LIN {X 0,Y 523.912,Z 870.031,A -85,B 0,C 180,E1 -4697.971,E2 -4697.971} C_VEL
LIN {X 0,Y 523.923,Z 870.031,A -85,B 0,C 180,E1 -4700.412,E2 -4700.412} C_VEL
LIN {X 0,Y 523.884,Z 870.04,A -85,B 0,C 180,E1 -4702.895,E2 -4702.895} C_VEL
LIN {X 0,Y 523.871,Z 870.043,A -85,B 0,C 180,E1 -4705.423,E2 -4705.423} C_VEL
LIN {X 0,Y 523.896,Z 870.034,A -85,B 0,C 180,E1 -4708.003,E2 -4708.003} C_VEL
LIN {X 0,Y 523.895,Z 870.034,A -85,B 0,C 180,E1 -4710.845,E2 -4710.845} C_VEL
LIN {X 0,Y 523.911,Z 870.039,A -85,B 0,C 180,E1 -4713.726,E2 -4713.726} C_VEL
LIN {X 0,Y 523.854,Z 870.039,A -85,B 0,C 180,E1 -4716.393,E2 -4716.393} C_VEL
LIN {X 0,Y 523.886,Z 870.034,A -85,B 0,C 180,E1 -4719.088,E2 -4719.088} C_VEL
LIN {X 0,Y 523.885,Z 870.042,A -85,B 0,C 180,E1 -4722.125,E2 -4722.125} C_VEL
LIN {X 0,Y 523.93,Z 870.029,A -85,B 0,C 180,E1 -4725.311,E2 -4725.311} C_VEL
LIN {X 0,Y 523.875,Z 870.039,A -85,B 0,C 180,E1 -4728.7,E2 -4728.7} C_VEL
LIN {X 0,Y 523.872,Z 870.038,A -85,B 0,C 180,E1 -4731.894,E2 -4731.894} C_VEL
LIN {X 0,Y 523.912,Z 870.035,A -85,B 0,C 180,E1 -4734.913,E2 -4734.913} C_VEL
LIN {X 0,Y 523.899,Z 870.032,A -85,B 0,C 180,E1 -4737.686,E2 -4737.686} C_VEL
LIN {X 0,Y 523.864,Z 870.039,A -85,B 0,C 180,E1 -4740.239,E2 -4740.239} C_VEL
LIN {X 0,Y 523.889,Z 870.043,A -85,B 0,C 180,E1 -4742.863,E2 -4742.863} C_VEL
LIN {X 0,Y 523.909,Z 870.036,A -85,B 0,C 180,E1 -4745.809,E2 -4745.809} C_VEL
LIN {X 0,Y 523.951,Z 870.114,A -85,B 0,C 180,E1 -4746.821,E2 -4746.821} C_VEL
LIN {X 0,Y 525.037,Z 877.349,A -85,B 0,C 180,E1 -4748.194,E2 -4748.194} C_VEL
LIN {X 0,Y 524.713,Z 893.158,A -85,B 0,C 180,E1 -4751.046,E2 -4751.046} C_VEL
LIN {X 0,Y 524.282,Z 909.934,A -85,B 0,C 180,E1 -4754.05,E2 -4754.05} C_VEL
LIN {X 0,Y 523.984,Z 926.682,A -85,B 0,C 180,E1 -4757.017,E2 -4757.017} C_VEL
LIN {X 0,Y 523.894,Z 932.763,A -85,B 0,C 180,E1 -4758.086,E2 -4758.086} C_VEL
LIN {X 0,Y 524.95,Z 941.667,A -85,B 0,C 180,E1 -4758.233,E2 -4758.233} C_VEL
LIN {X 0,Y 524.777,Z 1009.129,A -85,B 0,C 180,E1 -4759.169,E2 -4759.169} C_VEL
LIN {X 0,Y 524.62,Z 1018.404,A -85,B 0,C 180,E1 -4759.385,E2 -4759.385} C_VEL
LIN {X 0,Y 524.516,Z 1026.88,A -85,B 0,C 180,E1 -4759.676,E2 -4759.676} C_VEL
LIN {X 0,Y 524.389,Z 1035.388,A -85,B 0,C 180,E1 -4760.063,E2 -4760.063} C_VEL
LIN {X 0,Y 524.242,Z 1043.722,A -85,B 0,C 180,E1 -4760.548,E2 -4760.548} C_VEL
LIN {X 0,Y 524.1,Z 1051.761,A -85,B 0,C 180,E1 -4761.129,E2 -4761.129} C_VEL
LIN {X 0,Y 523.896,Z 1060.43,A -85,B 0,C 180,E1 -4761.902,E2 -4761.902} C_VEL
LIN {X 0,Y 523.705,Z 1068.937,A -85,B 0,C 180,E1 -4762.869,E2 -4762.869} C_VEL
LIN {X 0,Y 523.627,Z 1075.609,A -85,B 0,C 180,E1 -4763.836,E2 -4763.836} C_VEL
LIN {X 0,Y 523.485,Z 1079.988,A -85,B 0,C 180,E1 -4764.607,E2 -4764.607} C_VEL
LIN {X 0,Y 523.469,Z 1085.148,A -85,B 0,C 180,E1 -4765.765,E2 -4765.765} C_VEL
LIN {X 0,Y 523.412,Z 1087.787,A -85,B 0,C 180,E1 -4766.536,E2 -4766.536} C_VEL
LIN {X 0,Y 523.336,Z 1090.682,A -85,B 0,C 180,E1 -4767.691,E2 -4767.691} C_VEL
LIN {X 0,Y 523.273,Z 1091.931,A -85,B 0,C 180,E1 -4768.461,E2 -4768.461} C_VEL
LIN {X 0,Y 523.246,Z 1092.708,A -85,B 0,C 180,E1 -4769.23,E2 -4769.23} C_VEL
LIN {X 0,Y 523.243,Z 1093,A -85,B 0,C 180,E1 -4770,E2 -4770} C_VEL
LIN {X 0,Y 523.246,Z 1092.707,A -85,B 0,C 180,E1 -4770.769,E2 -4770.769} C_VEL
LIN {X 0,Y 523.273,Z 1091.931,A -85,B 0,C 180,E1 -4771.539,E2 -4771.539} C_VEL
LIN {X 0,Y 523.335,Z 1090.681,A -85,B 0,C 180,E1 -4772.309,E2 -4772.309} C_VEL
LIN {X 0,Y 523.407,Z 1087.787,A -85,B 0,C 180,E1 -4773.464,E2 -4773.464} C_VEL
LIN {X 0,Y 523.472,Z 1085.149,A -85,B 0,C 180,E1 -4774.235,E2 -4774.235} C_VEL
LIN {X 0,Y 523.484,Z 1079.986,A -85,B 0,C 180,E1 -4775.392,E2 -4775.392} C_VEL
LIN {X 0,Y 523.667,Z 1073.736,A -85,B 0,C 180,E1 -4776.469,E2 -4776.469} C_VEL
LIN {X 0,Y 523.752,Z 1065.742,A -85,B 0,C 180,E1 -4777.517,E2 -4777.517} C_VEL
LIN {X 0,Y 523.93,Z 1058.402,A -85,B 0,C 180,E1 -4778.291,E2 -4778.291} C_VEL
LIN {X 0,Y 524.154,Z 1050.538,A -85,B 0,C 180,E1 -4778.967,E2 -4778.967} C_VEL
LIN {X 0,Y 524.246,Z 1042.226,A -85,B 0,C 180,E1 -4779.549,E2 -4779.549} C_VEL
LIN {X 0,Y 524.484,Z 1031.613,A -85,B 0,C 180,E1 -4780.129,E2 -4780.129} C_VEL
LIN {X 0,Y 524.584,Z 1020.08,A -85,B 0,C 180,E1 -4780.566,E2 -4780.566} C_VEL
LIN {X 0,Y 524.741,Z 1010.444,A -85,B 0,C 180,E1 -4780.807,E2 -4780.807} C_VEL
LIN {X 0,Y 524.94,Z 952.856,A -85,B 0,C 180,E1 -4781.614,E2 -4781.614} C_VEL
LIN {X 0,Y 524.776,Z 939.225,A -85,B 0,C 180,E1 -4781.804,E2 -4781.804} C_VEL
LIN {X 0,Y 523.913,Z 932.728,A -85,B 0,C 180,E1 -4781.92,E2 -4781.92} C_VEL
LIN {X 0,Y 524.196,Z 915.268,A -85,B 0,C 180,E1 -4785.001,E2 -4785.001} C_VEL
LIN {X 0,Y 524.626,Z 896.76,A -85,B 0,C 180,E1 -4788.309,E2 -4788.309} C_VEL
LIN {X 0,Y 524.982,Z 879.434,A -85,B 0,C 180,E1 -4791.395,E2 -4791.395} C_VEL
LIN {X 0,Y 524.731,Z 874.352,A -85,B 0,C 180,E1 -4792.321,E2 -4792.321} C_VEL
LIN {X 0,Y 523.943,Z 870.037,A -85,B 0,C 180,E1 -4793.153,E2 -4793.153} C_VEL
LIN {X 0,Y 523.876,Z 870.04,A -85,B 0,C 180,E1 -4796.277,E2 -4796.277} C_VEL
LIN {X 0,Y 523.869,Z 870.044,A -85,B 0,C 180,E1 -4798.879,E2 -4798.879} C_VEL
LIN {X 0,Y 523.902,Z 870.04,A -85,B 0,C 180,E1 -4801.545,E2 -4801.545} C_VEL
LIN {X 0,Y 523.908,Z 870.033,A -85,B 0,C 180,E1 -4804.292,E2 -4804.292} C_VEL
LIN {X 0,Y 523.845,Z 870.044,A -85,B 0,C 180,E1 -4807.137,E2 -4807.137} C_VEL
LIN {X 0,Y 523.88,Z 870.038,A -85,B 0,C 180,E1 -4810.122,E2 -4810.122} C_VEL
LIN {X 0,Y 523.869,Z 870.038,A -85,B 0,C 180,E1 -4813.172,E2 -4813.172} C_VEL
LIN {X 0,Y 523.912,Z 870.039,A -85,B 0,C 180,E1 -4815.769,E2 -4815.769} C_VEL
LIN {X 0,Y 523.851,Z 870.039,A -85,B 0,C 180,E1 -4818.899,E2 -4818.899} C_VEL
LIN {X 0,Y 523.871,Z 870.042,A -85,B 0,C 180,E1 -4821.895,E2 -4821.895} C_VEL
LIN {X 0,Y 523.911,Z 870.034,A -85,B 0,C 180,E1 -4824.913,E2 -4824.913} C_VEL
LIN {X 0,Y 523.898,Z 870.034,A -85,B 0,C 180,E1 -4827.686,E2 -4827.686} C_VEL
LIN {X 0,Y 523.863,Z 870.042,A -85,B 0,C 180,E1 -4830.239,E2 -4830.239} C_VEL
LIN {X 0,Y 523.888,Z 870.043,A -85,B 0,C 180,E1 -4832.864,E2 -4832.864} C_VEL
LIN {X 0,Y 523.899,Z 870.036,A -85,B 0,C 180,E1 -4835.812,E2 -4835.812} C_VEL
LIN {X 0,Y 523.914,Z 870.041,A -85,B 0,C 180,E1 -4838.766,E2 -4838.766} C_VEL
LIN {X 0,Y 523.915,Z 870.041,A -85,B 0,C 180,E1 -4841.22,E2 -4841.22} C_VEL
LIN {X 0,Y 523.957,Z 870.182,A -85,B 0,C 180,E1 -4842.311,E2 -4842.311} C_VEL
LIN {X 0,Y 523.897,Z 880.418,A -85,B 0,C 180,E1 -4844.783,E2 -4844.783} C_VEL
LIN {X 0,Y 523.686,Z 894.295,A -85,B 0,C 180,E1 -4848.063,E2 -4848.063} C_VEL
LIN {X 0,Y 523.712,Z 894.979,A -85,B 0,C 180,E1 -4848.158,E2 -4848.158} C_VEL
LIN {X 0,Y 524.962,Z 903.624,A -85,B 0,C 180,E1 -4848.305,E2 -4848.305} C_VEL
LIN {X 0,Y 524.729,Z 969.368,A -85,B 0,C 180,E1 -4849.217,E2 -4849.217} C_VEL
LIN {X 0,Y 524.665,Z 978.561,A -85,B 0,C 180,E1 -4849.436,E2 -4849.436} C_VEL
LIN {X 0,Y 524.486,Z 988.212,A -85,B 0,C 180,E1 -4849.773,E2 -4849.773} C_VEL
LIN {X 0,Y 524.359,Z 998.292,A -85,B 0,C 180,E1 -4850.258,E2 -4850.258} C_VEL
LIN {X 0,Y 524.191,Z 1008.741,A -85,B 0,C 180,E1 -4850.936,E2 -4850.936} C_VEL
LIN {X 0,Y 523.927,Z 1017.984,A -85,B 0,C 180,E1 -4851.709,E2 -4851.709} C_VEL
LIN {X 0,Y 523.774,Z 1025.419,A -85,B 0,C 180,E1 -4852.483,E2 -4852.483} C_VEL
LIN {X 0,Y 523.663,Z 1032.503,A -85,B 0,C 180,E1 -4853.4,E2 -4853.4} C_VEL
LIN {X 0,Y 523.545,Z 1038.794,A -85,B 0,C 180,E1 -4854.415,E2 -4854.415} C_VEL
LIN {X 0,Y 523.417,Z 1043.444,A -85,B 0,C 180,E1 -4855.379,E2 -4855.379} C_VEL
LIN {X 0,Y 523.408,Z 1047.699,A -85,B 0,C 180,E1 -4856.536,E2 -4856.536} C_VEL
LIN {X 0,Y 523.336,Z 1050.634,A -85,B 0,C 180,E1 -4857.691,E2 -4857.691} C_VEL
LIN {X 0,Y 523.273,Z 1051.934,A -85,B 0,C 180,E1 -4858.461,E2 -4858.461} C_VEL
LIN {X 0,Y 523.246,Z 1052.719,A -85,B 0,C 180,E1 -4859.231,E2 -4859.231} C_VEL
LIN {X 0,Y 523.244,Z 1052.997,A -85,B 0,C 180,E1 -4860,E2 -4860} C_VEL
LIN {X 0,Y 523.247,Z 1052.771,A -85,B 0,C 180,E1 -4860.77,E2 -4860.77} C_VEL
LIN {X 0,Y 523.274,Z 1052.046,A -85,B 0,C 180,E1 -4861.54,E2 -4861.54} C_VEL
LIN {X 0,Y 523.337,Z 1050.82,A -85,B 0,C 180,E1 -4862.309,E2 -4862.309} C_VEL
LIN {X 0,Y 523.406,Z 1047.96,A -85,B 0,C 180,E1 -4863.464,E2 -4863.464} C_VEL
LIN {X 0,Y 523.409,Z 1043.83,A -85,B 0,C 180,E1 -4864.621,E2 -4864.621} C_VEL
LIN {X 0,Y 523.606,Z 1038.224,A -85,B 0,C 180,E1 -4865.778,E2 -4865.778} C_VEL
LIN {X 0,Y 523.623,Z 1032.601,A -85,B 0,C 180,E1 -4866.676,E2 -4866.676} C_VEL
LIN {X 0,Y 523.789,Z 1024.48,A -85,B 0,C 180,E1 -4867.711,E2 -4867.711} C_VEL
LIN {X 0,Y 523.987,Z 1015.836,A -85,B 0,C 180,E1 -4868.582,E2 -4868.582} C_VEL
LIN {X 0,Y 524.228,Z 1005.965,A -85,B 0,C 180,E1 -4869.355,E2 -4869.355} C_VEL
LIN {X 0,Y 524.376,Z 996.263,A -85,B 0,C 180,E1 -4869.937,E2 -4869.937} C_VEL
LIN {X 0,Y 524.486,Z 988.005,A -85,B 0,C 180,E1 -4870.325,E2 -4870.325} C_VEL
LIN {X 0,Y 524.604,Z 979.109,A -85,B 0,C 180,E1 -4870.64,E2 -4870.64} C_VEL
LIN {X 0,Y 524.761,Z 970.227,A -85,B 0,C 180,E1 -4870.856,E2 -4870.856} C_VEL
LIN {X 0,Y 524.819,Z 902.474,A -85,B 0,C 180,E1 -4871.804,E2 -4871.804} C_VEL
LIN {X 0,Y 523.675,Z 894.664,A -85,B 0,C 180,E1 -4871.941,E2 -4871.941} C_VEL
LIN {X 0,Y 523.898,Z 880.793,A -85,B 0,C 180,E1 -4875.217,E2 -4875.217} C_VEL
LIN {X 0,Y 524.012,Z 870.024,A -85,B 0,C 180,E1 -4877.816,E2 -4877.816} C_VEL
LIN {X 0,Y 523.916,Z 870.038,A -85,B 0,C 180,E1 -4881.235,E2 -4881.235} C_VEL
LIN {X 0,Y 523.898,Z 870.034,A -85,B 0,C 180,E1 -4884.574,E2 -4884.574} C_VEL
LIN {X 0,Y 523.913,Z 870.036,A -85,B 0,C 180,E1 -4887.705,E2 -4887.705} C_VEL
LIN {X 0,Y 523.899,Z 870.034,A -85,B 0,C 180,E1 -4890.846,E2 -4890.846} C_VEL
LIN {X 0,Y 523.927,Z 870.037,A -85,B 0,C 180,E1 -4893.729,E2 -4893.729} C_VEL
LIN {X 0,Y 523.856,Z 870.04,A -85,B 0,C 180,E1 -4896.279,E2 -4896.279} C_VEL
LIN {X 0,Y 523.205,Z 870.12,A -85,B 0,C 180,E1 -4896.921,E2 -4896.921} C_VEL
LIN {X 0,Y 520.366,Z 870.48,A -85,B 0,C 180,E1 -4897.963,E2 -4897.963} C_VEL
LIN {X 0,Y 517.955,Z 870.776,A -85,B 0,C 180,E1 -4898.802,E2 -4898.802} C_VEL
LIN {X 0,Y 516.915,Z 870.906,A -85,B 0,C 180,E1 -4899.45,E2 -4899.45} C_VEL
LIN {X 0,Y 516.829,Z 870.919,A -85,B 0,C 180,E1 -4899.669,E2 -4899.669} C_VEL
LIN {X 0,Y 516.843,Z 870.912,A -85,B 0,C 180,E1 -4902.836,E2 -4902.836} C_VEL
LIN {X 0,Y 516.899,Z 870.905,A -85,B 0,C 180,E1 -4905.007,E2 -4905.007} C_VEL
LIN {X 0,Y 516.831,Z 870.921,A -85,B 0,C 180,E1 -4908.41,E2 -4908.41} C_VEL
LIN {X 0,Y 516.855,Z 870.91,A -85,B 0,C 180,E1 -4911.282,E2 -4911.282} C_VEL
LIN {X 0,Y 516.853,Z 870.918,A -85,B 0,C 180,E1 -4914.674,E2 -4914.674} C_VEL
LIN {X 0,Y 516.87,Z 870.909,A -85,B 0,C 180,E1 -4917.462,E2 -4917.462} C_VEL
LIN {X 0,Y 516.841,Z 870.916,A -85,B 0,C 180,E1 -4920.491,E2 -4920.491} C_VEL
LIN {X 0,Y 516.83,Z 870.917,A -85,B 0,C 180,E1 -4923.337,E2 -4923.337} C_VEL
LIN {X 0,Y 516.871,Z 870.908,A -85,B 0,C 180,E1 -4925.926,E2 -4925.926} C_VEL
LIN {X 0,Y 516.869,Z 870.909,A -85,B 0,C 180,E1 -4928.462,E2 -4928.462} C_VEL
LIN {X 0,Y 516.871,Z 870.912,A -85,B 0,C 180,E1 -4930.954,E2 -4930.954} C_VEL
LIN {X 0,Y 516.876,Z 870.917,A -85,B 0,C 180,E1 -4933.409,E2 -4933.409} C_VEL
LIN {X 0,Y 516.875,Z 870.912,A -85,B 0,C 180,E1 -4935.833,E2 -4935.833} C_VEL
LIN {X 0,Y 516.925,Z 870.903,A -85,B 0,C 180,E1 -4938.233,E2 -4938.233} C_VEL
LIN {X 0,Y 516.921,Z 870.906,A -85,B 0,C 180,E1 -4941.399,E2 -4941.399} C_VEL
LIN {X 0,Y 516.981,Z 870.896,A -85,B 0,C 180,E1 -4944.54,E2 -4944.54} C_VEL
LIN {X 0,Y 517.071,Z 870.887,A -85,B 0,C 180,E1 -4947.663,E2 -4947.663} C_VEL
LIN {X 0,Y 517.068,Z 870.891,A -85,B 0,C 180,E1 -4950,E2 -4950} C_VEL
LIN {X 0,Y 517.068,Z 870.891,A -85,B 0,C 180,E1 -4952.337,E2 -4952.337} C_VEL
LIN {X 0,Y 516.97,Z 870.903,A -85,B 0,C 180,E1 -4956.244,E2 -4956.244} C_VEL
LIN {X 0,Y 516.905,Z 870.904,A -85,B 0,C 180,E1 -4959.39,E2 -4959.39} C_VEL
LIN {X 0,Y 516.884,Z 870.914,A -85,B 0,C 180,E1 -4962.565,E2 -4962.565} C_VEL
LIN {X 0,Y 516.838,Z 870.912,A -85,B 0,C 180,E1 -4965.781,E2 -4965.781} C_VEL
LIN {X 0,Y 516.875,Z 870.908,A -85,B 0,C 180,E1 -4968.224,E2 -4968.224} C_VEL
LIN {X 0,Y 516.882,Z 870.911,A -85,B 0,C 180,E1 -4970.703,E2 -4970.703} C_VEL
LIN {X 0,Y 516.841,Z 870.92,A -85,B 0,C 180,E1 -4973.225,E2 -4973.225} C_VEL
LIN {X 0,Y 516.861,Z 870.909,A -85,B 0,C 180,E1 -4976.176,E2 -4976.176} C_VEL
LIN {X 0,Y 516.833,Z 870.913,A -85,B 0,C 180,E1 -4978.421,E2 -4978.421} C_VEL
LIN {X 0,Y 516.849,Z 870.914,A -85,B 0,C 180,E1 -4981.112,E2 -4981.112} C_VEL
LIN {X 0,Y 516.873,Z 870.913,A -85,B 0,C 180,E1 -4983.959,E2 -4983.959} C_VEL
LIN {X 0,Y 516.799,Z 870.917,A -85,B 0,C 180,E1 -4986.753,E2 -4986.753} C_VEL
LIN {X 0,Y 516.827,Z 870.921,A -85,B 0,C 180,E1 -4989.727,E2 -4989.727} C_VEL
LIN {X 0,Y 516.841,Z 870.912,A -85,B 0,C 180,E1 -4992.836,E2 -4992.836} C_VEL
LIN {X 0,Y 516.901,Z 870.904,A -85,B 0,C 180,E1 -4995.007,E2 -4995.007} C_VEL
LIN {X 0,Y 516.832,Z 870.92,A -85,B 0,C 180,E1 -4998.409,E2 -4998.409} C_VEL
LIN {X 0,Y 516.854,Z 870.91,A -85,B 0,C 180,E1 -5001.281,E2 -5001.281} C_VEL
LIN {X 0,Y 516.852,Z 870.918,A -85,B 0,C 180,E1 -5004.673,E2 -5004.673} C_VEL
LIN {X 0,Y 516.871,Z 870.909,A -85,B 0,C 180,E1 -5007.462,E2 -5007.462} C_VEL
LIN {X 0,Y 516.841,Z 870.916,A -85,B 0,C 180,E1 -5010.491,E2 -5010.491} C_VEL
LIN {X 0,Y 516.83,Z 870.917,A -85,B 0,C 180,E1 -5013.336,E2 -5013.336} C_VEL
LIN {X 0,Y 516.871,Z 870.908,A -85,B 0,C 180,E1 -5015.926,E2 -5015.926} C_VEL
LIN {X 0,Y 516.869,Z 870.909,A -85,B 0,C 180,E1 -5018.461,E2 -5018.461} C_VEL
LIN {X 0,Y 516.87,Z 870.913,A -85,B 0,C 180,E1 -5020.953,E2 -5020.953} C_VEL
LIN {X 0,Y 516.874,Z 870.917,A -85,B 0,C 180,E1 -5023.408,E2 -5023.408} C_VEL
LIN {X 0,Y 516.867,Z 870.913,A -85,B 0,C 180,E1 -5025.832,E2 -5025.832} C_VEL
LIN {X 0,Y 516.923,Z 870.903,A -85,B 0,C 180,E1 -5028.232,E2 -5028.232} C_VEL
LIN {X 0,Y 516.919,Z 870.906,A -85,B 0,C 180,E1 -5031.398,E2 -5031.398} C_VEL
LIN {X 0,Y 516.979,Z 870.896,A -85,B 0,C 180,E1 -5034.539,E2 -5034.539} C_VEL
LIN {X 0,Y 517.069,Z 870.888,A -85,B 0,C 180,E1 -5037.663,E2 -5037.663} C_VEL
LIN {X 0,Y 517.066,Z 870.892,A -85,B 0,C 180,E1 -5040,E2 -5040} C_VEL
LIN {X 0,Y 517.066,Z 870.891,A -85,B 0,C 180,E1 -5042.337,E2 -5042.337} C_VEL
LIN {X 0,Y 516.968,Z 870.903,A -85,B 0,C 180,E1 -5046.243,E2 -5046.243} C_VEL
LIN {X 0,Y 516.902,Z 870.904,A -85,B 0,C 180,E1 -5049.39,E2 -5049.39} C_VEL
LIN {X 0,Y 516.882,Z 870.915,A -85,B 0,C 180,E1 -5052.565,E2 -5052.565} C_VEL
LIN {X 0,Y 516.904,Z 870.908,A -85,B 0,C 180,E1 -5055.128,E2 -5055.128} C_VEL
LIN {X 0,Y 516.871,Z 870.909,A -85,B 0,C 180,E1 -5058.224,E2 -5058.224} C_VEL
LIN {X 0,Y 516.879,Z 870.912,A -85,B 0,C 180,E1 -5060.703,E2 -5060.703} C_VEL
LIN {X 0,Y 516.837,Z 870.921,A -85,B 0,C 180,E1 -5063.225,E2 -5063.225} C_VEL
LIN {X 0,Y 516.857,Z 870.91,A -85,B 0,C 180,E1 -5066.176,E2 -5066.176} C_VEL
LIN {X 0,Y 516.829,Z 870.913,A -85,B 0,C 180,E1 -5068.42,E2 -5068.42} C_VEL
LIN {X 0,Y 516.845,Z 870.915,A -85,B 0,C 180,E1 -5071.112,E2 -5071.112} C_VEL
LIN {X 0,Y 516.869,Z 870.913,A -85,B 0,C 180,E1 -5073.959,E2 -5073.959} C_VEL
LIN {X 0,Y 516.795,Z 870.917,A -85,B 0,C 180,E1 -5076.753,E2 -5076.753} C_VEL
LIN {X 0,Y 516.823,Z 870.922,A -85,B 0,C 180,E1 -5079.727,E2 -5079.727} C_VEL
LIN {X 0,Y 516.836,Z 870.913,A -85,B 0,C 180,E1 -5082.836,E2 -5082.836} C_VEL
LIN {X 0,Y 516.896,Z 870.905,A -85,B 0,C 180,E1 -5085.007,E2 -5085.007} C_VEL
LIN {X 0,Y 516.828,Z 870.92,A -85,B 0,C 180,E1 -5088.409,E2 -5088.409} C_VEL
LIN {X 0,Y 516.85,Z 870.911,A -85,B 0,C 180,E1 -5091.281,E2 -5091.281} C_VEL
LIN {X 0,Y 516.848,Z 870.918,A -85,B 0,C 180,E1 -5094.673,E2 -5094.673} C_VEL
LIN {X 0,Y 516.866,Z 870.909,A -85,B 0,C 180,E1 -5097.462,E2 -5097.462} C_VEL
LIN {X 0,Y 516.837,Z 870.917,A -85,B 0,C 180,E1 -5100.491,E2 -5100.491} C_VEL
LIN {X 0,Y 516.825,Z 870.921,A -85,B 0,C 180,E1 -5103.336,E2 -5103.336} C_VEL
LIN {X 0,Y 516.904,Z 870.951,A -85,B 0,C 180,E1 -5106.672,E2 -5106.672} C_VEL
LIN {X 0,Y 518.076,Z 878.33,A -85,B 0,C 180,E1 -5108.096,E2 -5108.096} C_VEL
LIN {X 0,Y 517.716,Z 894.138,A -85,B 0,C 180,E1 -5110.986,E2 -5110.986} C_VEL
LIN {X 0,Y 517.268,Z 912.167,A -85,B 0,C 180,E1 -5114.232,E2 -5114.232} C_VEL
LIN {X 0,Y 516.888,Z 930.032,A -85,B 0,C 180,E1 -5117.435,E2 -5117.435} C_VEL
LIN {X 0,Y 516.861,Z 932.914,A -85,B 0,C 180,E1 -5117.924,E2 -5117.924} C_VEL
LIN {X 0,Y 517.983,Z 941.173,A -85,B 0,C 180,E1 -5118.066,E2 -5118.066} C_VEL
LIN {X 0,Y 517.827,Z 1009.137,A -85,B 0,C 180,E1 -5119.022,E2 -5119.022} C_VEL
LIN {X 0,Y 517.654,Z 1018.404,A -85,B 0,C 180,E1 -5119.241,E2 -5119.241} C_VEL
LIN {X 0,Y 517.534,Z 1026.879,A -85,B 0,C 180,E1 -5119.535,E2 -5119.535} C_VEL
LIN {X 0,Y 517.4,Z 1035.386,A -85,B 0,C 180,E1 -5119.928,E2 -5119.928} C_VEL
LIN {X 0,Y 517.25,Z 1043.72,A -85,B 0,C 180,E1 -5120.419,E2 -5120.419} C_VEL
LIN {X 0,Y 517.098,Z 1051.759,A -85,B 0,C 180,E1 -5121.008,E2 -5121.008} C_VEL
LIN {X 0,Y 516.843,Z 1060.431,A -85,B 0,C 180,E1 -5121.791,E2 -5121.791} C_VEL
LIN {X 0,Y 516.655,Z 1068.937,A -85,B 0,C 180,E1 -5122.771,E2 -5122.771} C_VEL
LIN {X 0,Y 516.561,Z 1075.609,A -85,B 0,C 180,E1 -5123.751,E2 -5123.751} C_VEL
LIN {X 0,Y 516.431,Z 1079.988,A -85,B 0,C 180,E1 -5124.533,E2 -5124.533} C_VEL
LIN {X 0,Y 516.392,Z 1085.148,A -85,B 0,C 180,E1 -5125.707,E2 -5125.707} C_VEL
LIN {X 0,Y 516.329,Z 1087.787,A -85,B 0,C 180,E1 -5126.488,E2 -5126.488} C_VEL
LIN {X 0,Y 516.262,Z 1090.681,A -85,B 0,C 180,E1 -5127.659,E2 -5127.659} C_VEL
LIN {X 0,Y 516.19,Z 1091.93,A -85,B 0,C 180,E1 -5128.439,E2 -5128.439} C_VEL
LIN {X 0,Y 516.156,Z 1092.707,A -85,B 0,C 180,E1 -5129.22,E2 -5129.22} C_VEL
LIN {X 0,Y 516.151,Z 1093,A -85,B 0,C 180,E1 -5130,E2 -5130} C_VEL
LIN {X 0,Y 516.156,Z 1092.707,A -85,B 0,C 180,E1 -5130.78,E2 -5130.78} C_VEL
LIN {X 0,Y 516.19,Z 1091.93,A -85,B 0,C 180,E1 -5131.56,E2 -5131.56} C_VEL
LIN {X 0,Y 516.262,Z 1090.681,A -85,B 0,C 180,E1 -5132.34,E2 -5132.34} C_VEL
LIN {X 0,Y 516.325,Z 1087.787,A -85,B 0,C 180,E1 -5133.512,E2 -5133.512} C_VEL
LIN {X 0,Y 516.394,Z 1085.149,A -85,B 0,C 180,E1 -5134.293,E2 -5134.293} C_VEL
LIN {X 0,Y 516.431,Z 1079.986,A -85,B 0,C 180,E1 -5135.466,E2 -5135.466} C_VEL
LIN {X 0,Y 516.58,Z 1074.231,A -85,B 0,C 180,E1 -5136.478,E2 -5136.478} C_VEL
LIN {X 0,Y 516.683,Z 1067.436,A -85,B 0,C 180,E1 -5137.424,E2 -5137.424} C_VEL
LIN {X 0,Y 516.862,Z 1059.421,A -85,B 0,C 180,E1 -5138.307,E2 -5138.307} C_VEL
LIN {X 0,Y 517.07,Z 1051.767,A -85,B 0,C 180,E1 -5138.993,E2 -5138.993} C_VEL
LIN {X 0,Y 517.226,Z 1043.725,A -85,B 0,C 180,E1 -5139.581,E2 -5139.581} C_VEL
LIN {X 0,Y 517.399,Z 1035.393,A -85,B 0,C 180,E1 -5140.072,E2 -5140.072} C_VEL
LIN {X 0,Y 517.533,Z 1026.89,A -85,B 0,C 180,E1 -5140.465,E2 -5140.465} C_VEL
LIN {X 0,Y 517.689,Z 1016.753,A -85,B 0,C 180,E1 -5140.808,E2 -5140.808} C_VEL
LIN {X 0,Y 517.871,Z 1005.092,A -85,B 0,C 180,E1 -5141.051,E2 -5141.051} C_VEL
LIN {X 0,Y 517.887,Z 940.331,A -85,B 0,C 180,E1 -5141.948,E2 -5141.948} C_VEL
LIN {X 0,Y 516.853,Z 932.68,A -85,B 0,C 180,E1 -5142.093,E2 -5142.093} C_VEL
LIN {X 0,Y 517.199,Z 915.041,A -85,B 0,C 180,E1 -5145.25,E2 -5145.25} C_VEL
LIN {X 0,Y 517.609,Z 897.395,A -85,B 0,C 180,E1 -5148.402,E2 -5148.402} C_VEL
LIN {X 0,Y 517.903,Z 882.556,A -85,B 0,C 180,E1 -5151.076,E2 -5151.076} C_VEL
LIN {X 0,Y 517.904,Z 876.83,A -85,B 0,C 180,E1 -5152.121,E2 -5152.121} C_VEL
LIN {X 0,Y 516.884,Z 870.915,A -85,B 0,C 180,E1 -5153.276,E2 -5153.276} C_VEL
LIN {X 0,Y 516.824,Z 870.921,A -85,B 0,C 180,E1 -5156.663,E2 -5156.663} C_VEL
LIN {X 0,Y 516.835,Z 870.919,A -85,B 0,C 180,E1 -5159.509,E2 -5159.509} C_VEL
LIN {X 0,Y 516.864,Z 870.911,A -85,B 0,C 180,E1 -5162.538,E2 -5162.538} C_VEL
LIN {X 0,Y 516.846,Z 870.92,A -85,B 0,C 180,E1 -5165.327,E2 -5165.327} C_VEL
LIN {X 0,Y 516.848,Z 870.912,A -85,B 0,C 180,E1 -5168.719,E2 -5168.719} C_VEL
LIN {X 0,Y 516.828,Z 870.922,A -85,B 0,C 180,E1 -5171.784,E2 -5171.784} C_VEL
LIN {X 0,Y 516.894,Z 870.906,A -85,B 0,C 180,E1 -5175.007,E2 -5175.007} C_VEL
LIN {X 0,Y 516.827,Z 870.919,A -85,B 0,C 180,E1 -5178.41,E2 -5178.41} C_VEL
LIN {X 0,Y 516.849,Z 870.912,A -85,B 0,C 180,E1 -5181.282,E2 -5181.282} C_VEL
LIN {X 0,Y 516.847,Z 870.917,A -85,B 0,C 180,E1 -5184.674,E2 -5184.674} C_VEL
LIN {X 0,Y 516.865,Z 870.91,A -85,B 0,C 180,E1 -5187.462,E2 -5187.462} C_VEL
LIN {X 0,Y 516.836,Z 870.922,A -85,B 0,C 180,E1 -5190.491,E2 -5190.491} C_VEL
LIN {X 0,Y 516.824,Z 870.917,A -85,B 0,C 180,E1 -5193.337,E2 -5193.337} C_VEL
LIN {X 0,Y 516.856,Z 870.914,A -85,B 0,C 180,E1 -5195.926,E2 -5195.926} C_VEL
LIN {X 0,Y 516.858,Z 870.916,A -85,B 0,C 180,E1 -5198.461,E2 -5198.461} C_VEL
LIN {X 0,Y 516.865,Z 870.919,A -85,B 0,C 180,E1 -5200.954,E2 -5200.954} C_VEL
LIN {X 0,Y 516.889,Z 870.978,A -85,B 0,C 180,E1 -5202.186,E2 -5202.186} C_VEL
LIN {X 0,Y 516.911,Z 877.482,A -85,B 0,C 180,E1 -5203.816,E2 -5203.816} C_VEL
LIN {X 0,Y 516.712,Z 888.994,A -85,B 0,C 180,E1 -5206.631,E2 -5206.631} C_VEL
LIN {X 0,Y 516.642,Z 894.642,A -85,B 0,C 180,E1 -5207.98,E2 -5207.98} C_VEL
LIN {X 0,Y 518.042,Z 905.254,A -85,B 0,C 180,E1 -5208.169,E2 -5208.169} C_VEL
LIN {X 0,Y 517.755,Z 969.401,A -85,B 0,C 180,E1 -5209.07,E2 -5209.07} C_VEL
LIN {X 0,Y 517.697,Z 978.581,A -85,B 0,C 180,E1 -5209.292,E2 -5209.292} C_VEL
LIN {X 0,Y 517.512,Z 988.225,A -85,B 0,C 180,E1 -5209.634,E2 -5209.634} C_VEL
LIN {X 0,Y 517.371,Z 998.307,A -85,B 0,C 180,E1 -5210.125,E2 -5210.125} C_VEL
LIN {X 0,Y 517.169,Z 1008.744,A -85,B 0,C 180,E1 -5210.812,E2 -5210.812} C_VEL
LIN {X 0,Y 516.894,Z 1017.992,A -85,B 0,C 180,E1 -5211.596,E2 -5211.596} C_VEL
LIN {X 0,Y 516.712,Z 1025.429,A -85,B 0,C 180,E1 -5212.38,E2 -5212.38} C_VEL
LIN {X 0,Y 516.621,Z 1032.128,A -85,B 0,C 180,E1 -5213.255,E2 -5213.255} C_VEL
LIN {X 0,Y 516.496,Z 1038.797,A -85,B 0,C 180,E1 -5214.339,E2 -5214.339} C_VEL
LIN {X 0,Y 516.322,Z 1043.444,A -85,B 0,C 180,E1 -5215.316,E2 -5215.316} C_VEL
LIN {X 0,Y 516.326,Z 1047.704,A -85,B 0,C 180,E1 -5216.489,E2 -5216.489} C_VEL
LIN {X 0,Y 516.263,Z 1050.639,A -85,B 0,C 180,E1 -5217.66,E2 -5217.66} C_VEL
LIN {X 0,Y 516.19,Z 1051.937,A -85,B 0,C 180,E1 -5218.44,E2 -5218.44} C_VEL
LIN {X 0,Y 516.157,Z 1052.719,A -85,B 0,C 180,E1 -5219.22,E2 -5219.22} C_VEL
LIN {X 0,Y 516.152,Z 1052.997,A -85,B 0,C 180,E1 -5220,E2 -5220} C_VEL
LIN {X 0,Y 516.157,Z 1052.774,A -85,B 0,C 180,E1 -5220.781,E2 -5220.781} C_VEL
LIN {X 0,Y 516.191,Z 1052.05,A -85,B 0,C 180,E1 -5221.561,E2 -5221.561} C_VEL
LIN {X 0,Y 516.263,Z 1050.823,A -85,B 0,C 180,E1 -5222.341,E2 -5222.341} C_VEL
LIN {X 0,Y 516.324,Z 1047.959,A -85,B 0,C 180,E1 -5223.512,E2 -5223.512} C_VEL
LIN {X 0,Y 516.315,Z 1043.825,A -85,B 0,C 180,E1 -5224.685,E2 -5224.685} C_VEL
LIN {X 0,Y 516.553,Z 1038.221,A -85,B 0,C 180,E1 -5225.857,E2 -5225.857} C_VEL
LIN {X 0,Y 516.585,Z 1031.97,A -85,B 0,C 180,E1 -5226.86,E2 -5226.86} C_VEL
LIN {X 0,Y 516.735,Z 1024.473,A -85,B 0,C 180,E1 -5227.817,E2 -5227.817} C_VEL
LIN {X 0,Y 516.972,Z 1015.828,A -85,B 0,C 180,E1 -5228.699,E2 -5228.699} C_VEL
LIN {X 0,Y 517.203,Z 1005.953,A -85,B 0,C 180,E1 -5229.484,E2 -5229.484} C_VEL
LIN {X 0,Y 517.382,Z 996.248,A -85,B 0,C 180,E1 -5230.073,E2 -5230.073} C_VEL
LIN {X 0,Y 517.514,Z 987.987,A -85,B 0,C 180,E1 -5230.466,E2 -5230.466} C_VEL
LIN {X 0,Y 517.649,Z 979.087,A -85,B 0,C 180,E1 -5230.784,E2 -5230.784} C_VEL
LIN {X 0,Y 517.809,Z 970.348,A -85,B 0,C 180,E1 -5231.001,E2 -5231.001} C_VEL
LIN {X 0,Y 517.901,Z 903.29,A -85,B 0,C 180,E1 -5231.952,E2 -5231.952} C_VEL
LIN {X 0,Y 516.624,Z 894.661,A -85,B 0,C 180,E1 -5232.106,E2 -5232.106} C_VEL
LIN {X 0,Y 516.875,Z 881.245,A -85,B 0,C 180,E1 -5235.336,E2 -5235.336} C_VEL
LIN {X 0,Y 516.954,Z 870.904,A -85,B 0,C 180,E1 -5237.889,E2 -5237.889} C_VEL
LIN {X 0,Y 516.879,Z 870.911,A -85,B 0,C 180,E1 -5240.703,E2 -5240.703} C_VEL
LIN {X 0,Y 516.84,Z 870.921,A -85,B 0,C 180,E1 -5243.225,E2 -5243.225} C_VEL
LIN {X 0,Y 516.861,Z 870.909,A -85,B 0,C 180,E1 -5246.177,E2 -5246.177} C_VEL
LIN {X 0,Y 516.83,Z 870.913,A -85,B 0,C 180,E1 -5248.421,E2 -5248.421} C_VEL
LIN {X 0,Y 516.849,Z 870.914,A -85,B 0,C 180,E1 -5251.113,E2 -5251.113} C_VEL
LIN {X 0,Y 516.882,Z 870.912,A -85,B 0,C 180,E1 -5253.962,E2 -5253.962} C_VEL
LIN {X 0,Y 516.807,Z 870.916,A -85,B 0,C 180,E1 -5256.752,E2 -5256.752} C_VEL
LIN {X 0,Y 516.829,Z 870.919,A -85,B 0,C 180,E1 -5259.669,E2 -5259.669} C_VEL
LIN {X 0,Y 516.16,Z 871.009,A -85,B 0,C 180,E1 -5260.32,E2 -5260.32} C_VEL
LIN {X 0,Y 513.312,Z 871.362,A -85,B 0,C 180,E1 -5261.377,E2 -5261.377} C_VEL
LIN {X 0,Y 510.907,Z 871.657,A -85,B 0,C 180,E1 -5262.228,E2 -5262.228} C_VEL
LIN {X 0,Y 509.873,Z 871.78,A -85,B 0,C 180,E1 -5262.885,E2 -5262.885} C_VEL
LIN {X 0,Y 509.787,Z 871.791,A -85,B 0,C 180,E1 -5263.108,E2 -5263.108} C_VEL
LIN {X 0,Y 509.809,Z 871.792,A -85,B 0,C 180,E1 -5265.796,E2 -5265.796} C_VEL
LIN {X 0,Y 509.785,Z 871.796,A -85,B 0,C 180,E1 -5268.567,E2 -5268.567} C_VEL
LIN {X 0,Y 509.806,Z 871.789,A -85,B 0,C 180,E1 -5271.794,E2 -5271.794} C_VEL
LIN {X 0,Y 509.81,Z 871.796,A -85,B 0,C 180,E1 -5274.62,E2 -5274.62} C_VEL
LIN {X 0,Y 509.838,Z 871.785,A -85,B 0,C 180,E1 -5277.479,E2 -5277.479} C_VEL
LIN {X 0,Y 509.788,Z 871.793,A -85,B 0,C 180,E1 -5280.289,E2 -5280.289} C_VEL
LIN {X 0,Y 509.816,Z 871.796,A -85,B 0,C 180,E1 -5282.94,E2 -5282.94} C_VEL
LIN {X 0,Y 509.822,Z 871.789,A -85,B 0,C 180,E1 -5285.572,E2 -5285.572} C_VEL
LIN {X 0,Y 509.813,Z 871.787,A -85,B 0,C 180,E1 -5288.148,E2 -5288.148} C_VEL
LIN {X 0,Y 509.832,Z 871.786,A -85,B 0,C 180,E1 -5290.68,E2 -5290.68} C_VEL
LIN {X 0,Y 509.849,Z 871.789,A -85,B 0,C 180,E1 -5293.174,E2 -5293.174} C_VEL
LIN {X 0,Y 509.849,Z 871.79,A -85,B 0,C 180,E1 -5295.634,E2 -5295.634} C_VEL
LIN {X 0,Y 509.859,Z 871.782,A -85,B 0,C 180,E1 -5298.873,E2 -5298.873} C_VEL
LIN {X 0,Y 509.878,Z 871.784,A -85,B 0,C 180,E1 -5302.077,E2 -5302.077} C_VEL
LIN {X 0,Y 509.937,Z 871.774,A -85,B 0,C 180,E1 -5304.464,E2 -5304.464} C_VEL
LIN {X 0,Y 510.038,Z 871.763,A -85,B 0,C 180,E1 -5307.631,E2 -5307.631} C_VEL
LIN {X 0,Y 510.037,Z 871.767,A -85,B 0,C 180,E1 -5310,E2 -5310} C_VEL
LIN {X 0,Y 510.036,Z 871.767,A -85,B 0,C 180,E1 -5312.369,E2 -5312.369} C_VEL
LIN {X 0,Y 509.936,Z 871.772,A -85,B 0,C 180,E1 -5315.536,E2 -5315.536} C_VEL
LIN {X 0,Y 509.879,Z 871.781,A -85,B 0,C 180,E1 -5317.923,E2 -5317.923} C_VEL
LIN {X 0,Y 509.86,Z 871.784,A -85,B 0,C 180,E1 -5321.127,E2 -5321.127} C_VEL
LIN {X 0,Y 509.819,Z 871.787,A -85,B 0,C 180,E1 -5323.553,E2 -5323.553} C_VEL
LIN {X 0,Y 509.806,Z 871.788,A -85,B 0,C 180,E1 -5326.005,E2 -5326.005} C_VEL
LIN {X 0,Y 509.831,Z 871.788,A -85,B 0,C 180,E1 -5328.485,E2 -5328.485} C_VEL
LIN {X 0,Y 509.828,Z 871.794,A -85,B 0,C 180,E1 -5331.003,E2 -5331.003} C_VEL
LIN {X 0,Y 509.801,Z 871.793,A -85,B 0,C 180,E1 -5333.565,E2 -5333.565} C_VEL
LIN {X 0,Y 509.801,Z 871.789,A -85,B 0,C 180,E1 -5336.352,E2 -5336.352} C_VEL
LIN {X 0,Y 509.797,Z 871.791,A -85,B 0,C 180,E1 -5338.849,E2 -5338.849} C_VEL
LIN {X 0,Y 509.785,Z 871.799,A -85,B 0,C 180,E1 -5341.593,E2 -5341.593} C_VEL
LIN {X 0,Y 509.826,Z 871.786,A -85,B 0,C 180,E1 -5344.416,E2 -5344.416} C_VEL
LIN {X 0,Y 509.762,Z 871.797,A -85,B 0,C 180,E1 -5347.346,E2 -5347.346} C_VEL
LIN {X 0,Y 509.79,Z 871.793,A -85,B 0,C 180,E1 -5350.387,E2 -5350.387} C_VEL
LIN {X 0,Y 509.795,Z 871.792,A -85,B 0,C 180,E1 -5353.575,E2 -5353.575} C_VEL
LIN {X 0,Y 509.795,Z 871.795,A -85,B 0,C 180,E1 -5356.425,E2 -5356.425} C_VEL
LIN {X 0,Y 509.789,Z 871.791,A -85,B 0,C 180,E1 -5359.612,E2 -5359.612} C_VEL
LIN {X 0,Y 509.762,Z 871.8,A -85,B 0,C 180,E1 -5362.654,E2 -5362.654} C_VEL
LIN {X 0,Y 509.842,Z 871.784,A -85,B 0,C 180,E1 -5365.8,E2 -5365.8} C_VEL
LIN {X 0,Y 509.818,Z 871.796,A -85,B 0,C 180,E1 -5368.726,E2 -5368.726} C_VEL
LIN {X 0,Y 509.826,Z 871.786,A -85,B 0,C 180,E1 -5372.05,E2 -5372.05} C_VEL
LIN {X 0,Y 509.785,Z 871.796,A -85,B 0,C 180,E1 -5374.699,E2 -5374.699} C_VEL
LIN {X 0,Y 509.828,Z 871.79,A -85,B 0,C 180,E1 -5377.459,E2 -5377.459} C_VEL
LIN {X 0,Y 509.848,Z 871.784,A -85,B 0,C 180,E1 -5379.841,E2 -5379.841} C_VEL
LIN {X 0,Y 509.848,Z 871.789,A -85,B 0,C 180,E1 -5383.173,E2 -5383.173} C_VEL
LIN {X 0,Y 509.834,Z 871.792,A -85,B 0,C 180,E1 -5385.633,E2 -5385.633} C_VEL
LIN {X 0,Y 509.891,Z 871.78,A -85,B 0,C 180,E1 -5388.131,E2 -5388.131} C_VEL
LIN {X 0,Y 509.872,Z 871.783,A -85,B 0,C 180,E1 -5391.279,E2 -5391.279} C_VEL
LIN {X 0,Y 509.919,Z 871.781,A -85,B 0,C 180,E1 -5393.669,E2 -5393.669} C_VEL
LIN {X 0,Y 509.858,Z 871.782,A -85,B 0,C 180,E1 -5396.839,E2 -5396.839} C_VEL
LIN {X 0,Y 509.922,Z 871.778,A -85,B 0,C 180,E1 -5398.42,E2 -5398.42} C_VEL
LIN {X 0,Y 510.035,Z 871.768,A -85,B 0,C 180,E1 -5400,E2 -5400} C_VEL
LIN {X 0,Y 510.034,Z 871.767,A -85,B 0,C 180,E1 -5402.369,E2 -5402.369} C_VEL
LIN {X 0,Y 509.934,Z 871.772,A -85,B 0,C 180,E1 -5405.536,E2 -5405.536} C_VEL
LIN {X 0,Y 509.876,Z 871.781,A -85,B 0,C 180,E1 -5407.922,E2 -5407.922} C_VEL
LIN {X 0,Y 509.857,Z 871.784,A -85,B 0,C 180,E1 -5411.126,E2 -5411.126} C_VEL
LIN {X 0,Y 509.823,Z 871.786,A -85,B 0,C 180,E1 -5413.553,E2 -5413.553} C_VEL
LIN {X 0,Y 509.805,Z 871.788,A -85,B 0,C 180,E1 -5416.004,E2 -5416.004} C_VEL
LIN {X 0,Y 509.828,Z 871.788,A -85,B 0,C 180,E1 -5418.485,E2 -5418.485} C_VEL
LIN {X 0,Y 509.824,Z 871.795,A -85,B 0,C 180,E1 -5421.002,E2 -5421.002} C_VEL
LIN {X 0,Y 509.798,Z 871.793,A -85,B 0,C 180,E1 -5423.565,E2 -5423.565} C_VEL
LIN {X 0,Y 509.798,Z 871.789,A -85,B 0,C 180,E1 -5426.352,E2 -5426.352} C_VEL
LIN {X 0,Y 509.793,Z 871.792,A -85,B 0,C 180,E1 -5428.849,E2 -5428.849} C_VEL
LIN {X 0,Y 509.781,Z 871.799,A -85,B 0,C 180,E1 -5431.593,E2 -5431.593} C_VEL
LIN {X 0,Y 509.821,Z 871.787,A -85,B 0,C 180,E1 -5434.415,E2 -5434.415} C_VEL
LIN {X 0,Y 509.759,Z 871.797,A -85,B 0,C 180,E1 -5437.345,E2 -5437.345} C_VEL
LIN {X 0,Y 509.785,Z 871.794,A -85,B 0,C 180,E1 -5440.387,E2 -5440.387} C_VEL
LIN {X 0,Y 509.79,Z 871.793,A -85,B 0,C 180,E1 -5443.575,E2 -5443.575} C_VEL
LIN {X 0,Y 509.79,Z 871.796,A -85,B 0,C 180,E1 -5446.425,E2 -5446.425} C_VEL
LIN {X 0,Y 509.785,Z 871.792,A -85,B 0,C 180,E1 -5449.612,E2 -5449.612} C_VEL
LIN {X 0,Y 509.757,Z 871.8,A -85,B 0,C 180,E1 -5452.654,E2 -5452.654} C_VEL
LIN {X 0,Y 509.837,Z 871.785,A -85,B 0,C 180,E1 -5455.8,E2 -5455.8} C_VEL
LIN {X 0,Y 509.814,Z 871.797,A -85,B 0,C 180,E1 -5458.726,E2 -5458.726} C_VEL
LIN {X 0,Y 509.821,Z 871.786,A -85,B 0,C 180,E1 -5462.05,E2 -5462.05} C_VEL
LIN {X 0,Y 509.781,Z 871.801,A -85,B 0,C 180,E1 -5464.699,E2 -5464.699} C_VEL
LIN {X 0,Y 509.865,Z 871.93,A -85,B 0,C 180,E1 -5466.546,E2 -5466.546} C_VEL
LIN {X 0,Y 511.078,Z 879.309,A -85,B 0,C 180,E1 -5467.993,E2 -5467.993} C_VEL
LIN {X 0,Y 510.724,Z 895.118,A -85,B 0,C 180,E1 -5470.924,E2 -5470.924} C_VEL
LIN {X 0,Y 510.253,Z 913.083,A -85,B 0,C 180,E1 -5474.202,E2 -5474.202} C_VEL
LIN {X 0,Y 509.837,Z 931.036,A -85,B 0,C 180,E1 -5477.44,E2 -5477.44} C_VEL
LIN {X 0,Y 509.803,Z 932.766,A -85,B 0,C 180,E1 -5477.752,E2 -5477.752} C_VEL
LIN {X 0,Y 511.064,Z 943.143,A -85,B 0,C 180,E1 -5477.929,E2 -5477.929} C_VEL
LIN {X 0,Y 510.881,Z 1009.214,A -85,B 0,C 180,E1 -5478.872,E2 -5478.872} C_VEL
LIN {X 0,Y 510.696,Z 1018.403,A -85,B 0,C 180,E1 -5479.092,E2 -5479.092} C_VEL
LIN {X 0,Y 510.567,Z 1026.878,A -85,B 0,C 180,E1 -5479.391,E2 -5479.391} C_VEL
LIN {X 0,Y 510.414,Z 1035.384,A -85,B 0,C 180,E1 -5479.789,E2 -5479.789} C_VEL
LIN {X 0,Y 510.258,Z 1043.719,A -85,B 0,C 180,E1 -5480.286,E2 -5480.286} C_VEL
LIN {X 0,Y 510.087,Z 1051.757,A -85,B 0,C 180,E1 -5480.883,E2 -5480.883} C_VEL
LIN {X 0,Y 509.819,Z 1060.431,A -85,B 0,C 180,E1 -5481.677,E2 -5481.677} C_VEL
LIN {X 0,Y 509.606,Z 1068.937,A -85,B 0,C 180,E1 -5482.671,E2 -5482.671} C_VEL
LIN {X 0,Y 509.492,Z 1075.609,A -85,B 0,C 180,E1 -5483.664,E2 -5483.664} C_VEL
LIN {X 0,Y 509.382,Z 1079.988,A -85,B 0,C 180,E1 -5484.458,E2 -5484.458} C_VEL
LIN {X 0,Y 509.298,Z 1085.149,A -85,B 0,C 180,E1 -5485.647,E2 -5485.647} C_VEL
LIN {X 0,Y 509.251,Z 1087.786,A -85,B 0,C 180,E1 -5486.439,E2 -5486.439} C_VEL
LIN {X 0,Y 509.191,Z 1090.68,A -85,B 0,C 180,E1 -5487.627,E2 -5487.627} C_VEL
LIN {X 0,Y 509.111,Z 1091.929,A -85,B 0,C 180,E1 -5488.418,E2 -5488.418} C_VEL
LIN {X 0,Y 509.07,Z 1092.706,A -85,B 0,C 180,E1 -5489.209,E2 -5489.209} C_VEL
LIN {X 0,Y 509.062,Z 1093,A -85,B 0,C 180,E1 -5490,E2 -5490} C_VEL
LIN {X 0,Y 509.07,Z 1092.706,A -85,B 0,C 180,E1 -5490.791,E2 -5490.791} C_VEL
LIN {X 0,Y 509.111,Z 1091.929,A -85,B 0,C 180,E1 -5491.582,E2 -5491.582} C_VEL
LIN {X 0,Y 509.191,Z 1090.68,A -85,B 0,C 180,E1 -5492.373,E2 -5492.373} C_VEL
LIN {X 0,Y 509.247,Z 1087.787,A -85,B 0,C 180,E1 -5493.56,E2 -5493.56} C_VEL
LIN {X 0,Y 509.3,Z 1085.149,A -85,B 0,C 180,E1 -5494.353,E2 -5494.353} C_VEL
LIN {X 0,Y 509.382,Z 1079.986,A -85,B 0,C 180,E1 -5495.542,E2 -5495.542} C_VEL
LIN {X 0,Y 509.493,Z 1074.853,A -85,B 0,C 180,E1 -5496.463,E2 -5496.463} C_VEL
LIN {X 0,Y 509.619,Z 1067.436,A -85,B 0,C 180,E1 -5497.528,E2 -5497.528} C_VEL
LIN {X 0,Y 509.843,Z 1059.42,A -85,B 0,C 180,E1 -5498.422,E2 -5498.422} C_VEL
LIN {X 0,Y 510.053,Z 1051.765,A -85,B 0,C 180,E1 -5499.117,E2 -5499.117} C_VEL
LIN {X 0,Y 510.233,Z 1043.724,A -85,B 0,C 180,E1 -5499.714,E2 -5499.714} C_VEL
LIN {X 0,Y 510.414,Z 1035.392,A -85,B 0,C 180,E1 -5500.211,E2 -5500.211} C_VEL
LIN {X 0,Y 510.564,Z 1026.888,A -85,B 0,C 180,E1 -5500.609,E2 -5500.609} C_VEL
LIN {X 0,Y 510.738,Z 1016.753,A -85,B 0,C 180,E1 -5500.957,E2 -5500.957} C_VEL
LIN {X 0,Y 510.923,Z 1005.447,A -85,B 0,C 180,E1 -5501.198,E2 -5501.198} C_VEL
LIN {X 0,Y 511.01,Z 941.466,A -85,B 0,C 180,E1 -5502.096,E2 -5502.096} C_VEL
LIN {X 0,Y 509.835,Z 932.658,A -85,B 0,C 180,E1 -5502.266,E2 -5502.266} C_VEL
LIN {X 0,Y 510.154,Z 915.431,A -85,B 0,C 180,E1 -5505.349,E2 -5505.349} C_VEL
LIN {X 0,Y 510.59,Z 898.205,A -85,B 0,C 180,E1 -5508.456,E2 -5508.456} C_VEL
LIN {X 0,Y 510.999,Z 881.106,A -85,B 0,C 180,E1 -5511.586,E2 -5511.586} C_VEL
LIN {X 0,Y 510.729,Z 876.511,A -85,B 0,C 180,E1 -5512.449,E2 -5512.449} C_VEL
LIN {X 0,Y 509.847,Z 871.791,A -85,B 0,C 180,E1 -5513.401,E2 -5513.401} C_VEL
LIN {X 0,Y 509.795,Z 871.795,A -85,B 0,C 180,E1 -5516.352,E2 -5516.352} C_VEL
LIN {X 0,Y 509.79,Z 871.798,A -85,B 0,C 180,E1 -5518.85,E2 -5518.85} C_VEL
LIN {X 0,Y 509.786,Z 871.798,A -85,B 0,C 180,E1 -5521.592,E2 -5521.592} C_VEL
LIN {X 0,Y 509.83,Z 871.787,A -85,B 0,C 180,E1 -5524.415,E2 -5524.415} C_VEL
LIN {X 0,Y 509.756,Z 871.802,A -85,B 0,C 180,E1 -5527.346,E2 -5527.346} C_VEL
LIN {X 0,Y 509.783,Z 871.792,A -85,B 0,C 180,E1 -5530.388,E2 -5530.388} C_VEL
LIN {X 0,Y 509.788,Z 871.797,A -85,B 0,C 180,E1 -5533.575,E2 -5533.575} C_VEL
LIN {X 0,Y 509.788,Z 871.794,A -85,B 0,C 180,E1 -5536.425,E2 -5536.425} C_VEL
LIN {X 0,Y 509.783,Z 871.794,A -85,B 0,C 180,E1 -5539.613,E2 -5539.613} C_VEL
LIN {X 0,Y 509.757,Z 871.799,A -85,B 0,C 180,E1 -5542.654,E2 -5542.654} C_VEL
LIN {X 0,Y 509.836,Z 871.787,A -85,B 0,C 180,E1 -5545.801,E2 -5545.801} C_VEL
LIN {X 0,Y 509.813,Z 871.795,A -85,B 0,C 180,E1 -5548.726,E2 -5548.726} C_VEL
LIN {X 0,Y 509.82,Z 871.789,A -85,B 0,C 180,E1 -5552.05,E2 -5552.05} C_VEL
LIN {X 0,Y 509.779,Z 871.802,A -85,B 0,C 180,E1 -5554.699,E2 -5554.699} C_VEL
LIN {X 0,Y 509.822,Z 871.792,A -85,B 0,C 180,E1 -5557.459,E2 -5557.459} C_VEL
LIN {X 0,Y 509.826,Z 871.793,A -85,B 0,C 180,E1 -5560.68,E2 -5560.68} C_VEL
LIN {X 0,Y 509.867,Z 871.826,A -85,B 0,C 180,E1 -5562.071,E2 -5562.071} C_VEL
LIN {X 0,Y 509.938,Z 877.806,A -85,B 0,C 180,E1 -5563.589,E2 -5563.589} C_VEL
LIN {X 0,Y 509.69,Z 889.236,A -85,B 0,C 180,E1 -5566.444,E2 -5566.444} C_VEL
LIN {X 0,Y 509.615,Z 894.776,A -85,B 0,C 180,E1 -5567.812,E2 -5567.812} C_VEL
LIN {X 0,Y 511.101,Z 905.25,A -85,B 0,C 180,E1 -5568.006,E2 -5568.006} C_VEL
LIN {X 0,Y 510.806,Z 969.433,A -85,B 0,C 180,E1 -5568.92,E2 -5568.92} C_VEL
LIN {X 0,Y 510.709,Z 978.601,A -85,B 0,C 180,E1 -5569.143,E2 -5569.143} C_VEL
LIN {X 0,Y 510.537,Z 988.239,A -85,B 0,C 180,E1 -5569.491,E2 -5569.491} C_VEL
LIN {X 0,Y 510.379,Z 998.323,A -85,B 0,C 180,E1 -5569.989,E2 -5569.989} C_VEL
LIN {X 0,Y 510.193,Z 1007.417,A -85,B 0,C 180,E1 -5570.586,E2 -5570.586} C_VEL
LIN {X 0,Y 509.898,Z 1016.996,A -85,B 0,C 180,E1 -5571.38,E2 -5571.38} C_VEL
LIN {X 0,Y 509.668,Z 1025.435,A -85,B 0,C 180,E1 -5572.274,E2 -5572.274} C_VEL
LIN {X 0,Y 509.544,Z 1032.756,A -85,B 0,C 180,E1 -5573.255,E2 -5573.255} C_VEL
LIN {X 0,Y 509.429,Z 1038.8,A -85,B 0,C 180,E1 -5574.26,E2 -5574.26} C_VEL
LIN {X 0,Y 509.235,Z 1043.444,A -85,B 0,C 180,E1 -5575.25,E2 -5575.25} C_VEL
LIN {X 0,Y 509.248,Z 1047.707,A -85,B 0,C 180,E1 -5576.44,E2 -5576.44} C_VEL
LIN {X 0,Y 509.192,Z 1050.642,A -85,B 0,C 180,E1 -5577.627,E2 -5577.627} C_VEL
LIN {X 0,Y 509.111,Z 1051.937,A -85,B 0,C 180,E1 -5578.418,E2 -5578.418} C_VEL
LIN {X 0,Y 509.07,Z 1052.718,A -85,B 0,C 180,E1 -5579.209,E2 -5579.209} C_VEL
LIN {X 0,Y 509.063,Z 1052.997,A -85,B 0,C 180,E1 -5580,E2 -5580} C_VEL
LIN {X 0,Y 509.071,Z 1052.776,A -85,B 0,C 180,E1 -5580.791,E2 -5580.791} C_VEL
LIN {X 0,Y 509.112,Z 1052.054,A -85,B 0,C 180,E1 -5581.582,E2 -5581.582} C_VEL
LIN {X 0,Y 509.192,Z 1050.826,A -85,B 0,C 180,E1 -5582.373,E2 -5582.373} C_VEL
LIN {X 0,Y 509.246,Z 1047.958,A -85,B 0,C 180,E1 -5583.561,E2 -5583.561} C_VEL
LIN {X 0,Y 509.228,Z 1043.819,A -85,B 0,C 180,E1 -5584.75,E2 -5584.75} C_VEL
LIN {X 0,Y 509.491,Z 1038.217,A -85,B 0,C 180,E1 -5585.939,E2 -5585.939} C_VEL
LIN {X 0,Y 509.523,Z 1031.888,A -85,B 0,C 180,E1 -5586.966,E2 -5586.966} C_VEL
LIN {X 0,Y 509.698,Z 1024.466,A -85,B 0,C 180,E1 -5587.926,E2 -5587.926} C_VEL
LIN {X 0,Y 509.944,Z 1015.819,A -85,B 0,C 180,E1 -5588.82,E2 -5588.82} C_VEL
LIN {X 0,Y 510.21,Z 1005.94,A -85,B 0,C 180,E1 -5589.615,E2 -5589.615} C_VEL
LIN {X 0,Y 510.397,Z 996.233,A -85,B 0,C 180,E1 -5590.212,E2 -5590.212} C_VEL
LIN {X 0,Y 510.547,Z 987.969,A -85,B 0,C 180,E1 -5590.61,E2 -5590.61} C_VEL
LIN {X 0,Y 510.702,Z 979.064,A -85,B 0,C 180,E1 -5590.933,E2 -5590.933} C_VEL
LIN {X 0,Y 510.857,Z 970.439,A -85,B 0,C 180,E1 -5591.15,E2 -5591.15} C_VEL
LIN {X 0,Y 510.932,Z 903.651,A -85,B 0,C 180,E1 -5592.111,E2 -5592.111} C_VEL
LIN {X 0,Y 509.593,Z 894.741,A -85,B 0,C 180,E1 -5592.276,E2 -5592.276} C_VEL
LIN {X 0,Y 509.848,Z 881.444,A -85,B 0,C 180,E1 -5595.552,E2 -5595.552} C_VEL
LIN {X 0,Y 509.919,Z 871.842,A -85,B 0,C 180,E1 -5597.931,E2 -5597.931} C_VEL
LIN {X 0,Y 509.824,Z 871.795,A -85,B 0,C 180,E1 -5601.003,E2 -5601.003} C_VEL
LIN {X 0,Y 509.803,Z 871.793,A -85,B 0,C 180,E1 -5603.565,E2 -5603.565} C_VEL
LIN {X 0,Y 509.802,Z 871.789,A -85,B 0,C 180,E1 -5606.353,E2 -5606.353} C_VEL
LIN {X 0,Y 509.794,Z 871.791,A -85,B 0,C 180,E1 -5608.85,E2 -5608.85} C_VEL
LIN {X 0,Y 509.79,Z 871.799,A -85,B 0,C 180,E1 -5611.593,E2 -5611.593} C_VEL
LIN {X 0,Y 509.834,Z 871.785,A -85,B 0,C 180,E1 -5614.415,E2 -5614.415} C_VEL
LIN {X 0,Y 509.777,Z 871.795,A -85,B 0,C 180,E1 -5617.345,E2 -5617.345} C_VEL
LIN {X 0,Y 509.788,Z 871.794,A -85,B 0,C 180,E1 -5620.388,E2 -5620.388} C_VEL
LIN {X 0,Y 509.787,Z 871.791,A -85,B 0,C 180,E1 -5623.108,E2 -5623.108} C_VEL
LIN {X 0,Y 509.112,Z 871.881,A -85,B 0,C 180,E1 -5623.768,E2 -5623.768} C_VEL
LIN {X 0,Y 506.242,Z 872.233,A -85,B 0,C 180,E1 -5624.838,E2 -5624.838} C_VEL
LIN {X 0,Y 503.83,Z 872.535,A -85,B 0,C 180,E1 -5625.701,E2 -5625.701} C_VEL
LIN {X 0,Y 502.812,Z 872.666,A -85,B 0,C 180,E1 -5626.368,E2 -5626.368} C_VEL
LIN {X 0,Y 502.739,Z 872.672,A -85,B 0,C 180,E1 -5626.593,E2 -5626.593} C_VEL
LIN {X 0,Y 502.752,Z 872.668,A -85,B 0,C 180,E1 -5629.015,E2 -5629.015} C_VEL
LIN {X 0,Y 502.753,Z 872.67,A -85,B 0,C 180,E1 -5632.043,E2 -5632.043} C_VEL
LIN {X 0,Y 502.785,Z 872.666,A -85,B 0,C 180,E1 -5635.033,E2 -5635.033} C_VEL
LIN {X 0,Y 502.761,Z 872.666,A -85,B 0,C 180,E1 -5637.914,E2 -5637.914} C_VEL
LIN {X 0,Y 502.755,Z 872.674,A -85,B 0,C 180,E1 -5640.708,E2 -5640.708} C_VEL
LIN {X 0,Y 502.773,Z 872.667,A -85,B 0,C 180,E1 -5643.461,E2 -5643.461} C_VEL
LIN {X 0,Y 502.757,Z 872.666,A -85,B 0,C 180,E1 -5646.085,E2 -5646.085} C_VEL
LIN {X 0,Y 502.771,Z 872.667,A -85,B 0,C 180,E1 -5648.688,E2 -5648.688} C_VEL
LIN {X 0,Y 502.798,Z 872.663,A -85,B 0,C 180,E1 -5651.897,E2 -5651.897} C_VEL
LIN {X 0,Y 502.84,Z 872.656,A -85,B 0,C 180,E1 -5654.665,E2 -5654.665} C_VEL
LIN {X 0,Y 502.844,Z 872.659,A -85,B 0,C 180,E1 -5658.06,E2 -5658.06} C_VEL
LIN {X 0,Y 502.837,Z 872.658,A -85,B 0,C 180,E1 -5661.156,E2 -5661.156} C_VEL
LIN {X 0,Y 502.872,Z 872.657,A -85,B 0,C 180,E1 -5663.581,E2 -5663.581} C_VEL
LIN {X 0,Y 502.738,Z 872.677,A -85,B 0,C 180,E1 -5665.992,E2 -5665.992} C_VEL
LIN {X 0,Y 503.005,Z 872.639,A -85,B 0,C 180,E1 -5667.598,E2 -5667.598} C_VEL
LIN {X 0,Y 503.006,Z 872.643,A -85,B 0,C 180,E1 -5670,E2 -5670} C_VEL
LIN {X 0,Y 503.003,Z 872.642,A -85,B 0,C 180,E1 -5672.402,E2 -5672.402} C_VEL
LIN {X 0,Y 502.893,Z 872.65,A -85,B 0,C 180,E1 -5675.614,E2 -5675.614} C_VEL
LIN {X 0,Y 502.85,Z 872.658,A -85,B 0,C 180,E1 -5678.034,E2 -5678.034} C_VEL
LIN {X 0,Y 502.837,Z 872.658,A -85,B 0,C 180,E1 -5681.284,E2 -5681.284} C_VEL
LIN {X 0,Y 502.8,Z 872.667,A -85,B 0,C 180,E1 -5684.572,E2 -5684.572} C_VEL
LIN {X 0,Y 502.795,Z 872.668,A -85,B 0,C 180,E1 -5687.07,E2 -5687.07} C_VEL
LIN {X 0,Y 502.779,Z 872.665,A -85,B 0,C 180,E1 -5689.602,E2 -5689.602} C_VEL
LIN {X 0,Y 502.786,Z 872.666,A -85,B 0,C 180,E1 -5692.696,E2 -5692.696} C_VEL
LIN {X 0,Y 502.762,Z 872.669,A -85,B 0,C 180,E1 -5695.68,E2 -5695.68} C_VEL
LIN {X 0,Y 502.764,Z 872.665,A -85,B 0,C 180,E1 -5698.378,E2 -5698.378} C_VEL
LIN {X 0,Y 502.765,Z 872.675,A -85,B 0,C 180,E1 -5701.492,E2 -5701.492} C_VEL
LIN {X 0,Y 502.778,Z 872.664,A -85,B 0,C 180,E1 -5704.439,E2 -5704.439} C_VEL
LIN {X 0,Y 502.719,Z 872.672,A -85,B 0,C 180,E1 -5707.168,E2 -5707.168} C_VEL
LIN {X 0,Y 502.733,Z 872.677,A -85,B 0,C 180,E1 -5710.021,E2 -5710.021} C_VEL
LIN {X 0,Y 502.741,Z 872.669,A -85,B 0,C 180,E1 -5713.235,E2 -5713.235} C_VEL
LIN {X 0,Y 502.771,Z 872.667,A -85,B 0,C 180,E1 -5715.658,E2 -5715.658} C_VEL
LIN {X 0,Y 502.753,Z 872.668,A -85,B 0,C 180,E1 -5719.014,E2 -5719.014} C_VEL
LIN {X 0,Y 502.747,Z 872.671,A -85,B 0,C 180,E1 -5722.041,E2 -5722.041} C_VEL
LIN {X 0,Y 502.785,Z 872.666,A -85,B 0,C 180,E1 -5725.032,E2 -5725.032} C_VEL
LIN {X 0,Y 502.761,Z 872.666,A -85,B 0,C 180,E1 -5727.913,E2 -5727.913} C_VEL
LIN {X 0,Y 502.756,Z 872.674,A -85,B 0,C 180,E1 -5730.707,E2 -5730.707} C_VEL
LIN {X 0,Y 502.773,Z 872.667,A -85,B 0,C 180,E1 -5733.461,E2 -5733.461} C_VEL
LIN {X 0,Y 502.757,Z 872.666,A -85,B 0,C 180,E1 -5736.084,E2 -5736.084} C_VEL
LIN {X 0,Y 502.77,Z 872.667,A -85,B 0,C 180,E1 -5738.688,E2 -5738.688} C_VEL
LIN {X 0,Y 502.797,Z 872.663,A -85,B 0,C 180,E1 -5741.897,E2 -5741.897} C_VEL
LIN {X 0,Y 502.827,Z 872.658,A -85,B 0,C 180,E1 -5744.67,E2 -5744.67} C_VEL
LIN {X 0,Y 502.843,Z 872.659,A -85,B 0,C 180,E1 -5748.06,E2 -5748.06} C_VEL
LIN {X 0,Y 502.835,Z 872.658,A -85,B 0,C 180,E1 -5751.156,E2 -5751.156} C_VEL
LIN {X 0,Y 502.87,Z 872.658,A -85,B 0,C 180,E1 -5753.58,E2 -5753.58} C_VEL
LIN {X 0,Y 502.734,Z 872.678,A -85,B 0,C 180,E1 -5755.991,E2 -5755.991} C_VEL
LIN {X 0,Y 503.003,Z 872.639,A -85,B 0,C 180,E1 -5757.597,E2 -5757.597} C_VEL
LIN {X 0,Y 503.004,Z 872.643,A -85,B 0,C 180,E1 -5760,E2 -5760} C_VEL
LIN {X 0,Y 503.001,Z 872.642,A -85,B 0,C 180,E1 -5762.402,E2 -5762.402} C_VEL
LIN {X 0,Y 502.891,Z 872.65,A -85,B 0,C 180,E1 -5765.614,E2 -5765.614} C_VEL
LIN {X 0,Y 502.848,Z 872.658,A -85,B 0,C 180,E1 -5768.034,E2 -5768.034} C_VEL
LIN {X 0,Y 502.834,Z 872.658,A -85,B 0,C 180,E1 -5771.284,E2 -5771.284} C_VEL
LIN {X 0,Y 502.813,Z 872.666,A -85,B 0,C 180,E1 -5774.571,E2 -5774.571} C_VEL
LIN {X 0,Y 502.786,Z 872.663,A -85,B 0,C 180,E1 -5777.909,E2 -5777.909} C_VEL
LIN {X 0,Y 502.804,Z 872.663,A -85,B 0,C 180,E1 -5780.527,E2 -5780.527} C_VEL
LIN {X 0,Y 502.778,Z 872.672,A -85,B 0,C 180,E1 -5783.041,E2 -5783.041} C_VEL
LIN {X 0,Y 502.758,Z 872.669,A -85,B 0,C 180,E1 -5785.68,E2 -5785.68} C_VEL
LIN {X 0,Y 502.76,Z 872.666,A -85,B 0,C 180,E1 -5788.377,E2 -5788.377} C_VEL
LIN {X 0,Y 502.761,Z 872.676,A -85,B 0,C 180,E1 -5791.492,E2 -5791.492} C_VEL
LIN {X 0,Y 502.774,Z 872.665,A -85,B 0,C 180,E1 -5794.438,E2 -5794.438} C_VEL
LIN {X 0,Y 502.716,Z 872.673,A -85,B 0,C 180,E1 -5797.168,E2 -5797.168} C_VEL
LIN {X 0,Y 502.729,Z 872.677,A -85,B 0,C 180,E1 -5800.021,E2 -5800.021} C_VEL
LIN {X 0,Y 502.736,Z 872.669,A -85,B 0,C 180,E1 -5803.235,E2 -5803.235} C_VEL
LIN {X 0,Y 502.766,Z 872.668,A -85,B 0,C 180,E1 -5805.658,E2 -5805.658} C_VEL
LIN {X 0,Y 502.749,Z 872.668,A -85,B 0,C 180,E1 -5809.014,E2 -5809.014} C_VEL
LIN {X 0,Y 502.742,Z 872.672,A -85,B 0,C 180,E1 -5812.041,E2 -5812.041} C_VEL
LIN {X 0,Y 502.781,Z 872.666,A -85,B 0,C 180,E1 -5815.032,E2 -5815.032} C_VEL
LIN {X 0,Y 502.756,Z 872.667,A -85,B 0,C 180,E1 -5817.913,E2 -5817.913} C_VEL
LIN {X 0,Y 502.751,Z 872.675,A -85,B 0,C 180,E1 -5820.707,E2 -5820.707} C_VEL
LIN {X 0,Y 502.768,Z 872.672,A -85,B 0,C 180,E1 -5823.461,E2 -5823.461} C_VEL
LIN {X 0,Y 502.834,Z 872.854,A -85,B 0,C 180,E1 -5826.416,E2 -5826.416} C_VEL
LIN {X 0,Y 504.102,Z 880.257,A -85,B 0,C 180,E1 -5827.887,E2 -5827.887} C_VEL
LIN {X 0,Y 503.735,Z 896.081,A -85,B 0,C 180,E1 -5830.86,E2 -5830.86} C_VEL
LIN {X 0,Y 503.202,Z 914.34,A -85,B 0,C 180,E1 -5834.237,E2 -5834.237} C_VEL
LIN {X 0,Y 502.78,Z 931.879,A -85,B 0,C 180,E1 -5837.446,E2 -5837.446} C_VEL
LIN {X 0,Y 502.754,Z 932.646,A -85,B 0,C 180,E1 -5837.585,E2 -5837.585} C_VEL
LIN {X 0,Y 504.109,Z 943.552,A -85,B 0,C 180,E1 -5837.774,E2 -5837.774} C_VEL
LIN {X 0,Y 503.906,Z 1008.798,A -85,B 0,C 180,E1 -5838.717,E2 -5838.717} C_VEL
LIN {X 0,Y 503.711,Z 1018.067,A -85,B 0,C 180,E1 -5838.939,E2 -5838.939} C_VEL
LIN {X 0,Y 503.606,Z 1026.635,A -85,B 0,C 180,E1 -5839.242,E2 -5839.242} C_VEL
LIN {X 0,Y 503.407,Z 1035.209,A -85,B 0,C 180,E1 -5839.645,E2 -5839.645} C_VEL
LIN {X 0,Y 503.243,Z 1043.607,A -85,B 0,C 180,E1 -5840.149,E2 -5840.149} C_VEL
LIN {X 0,Y 503.061,Z 1051.701,A -85,B 0,C 180,E1 -5840.755,E2 -5840.755} C_VEL
LIN {X 0,Y 502.815,Z 1059.397,A -85,B 0,C 180,E1 -5841.459,E2 -5841.459} C_VEL
LIN {X 0,Y 502.581,Z 1067.433,A -85,B 0,C 180,E1 -5842.366,E2 -5842.366} C_VEL
LIN {X 0,Y 502.462,Z 1073.744,A -85,B 0,C 180,E1 -5843.257,E2 -5843.257} C_VEL
LIN {X 0,Y 502.33,Z 1079.988,A -85,B 0,C 180,E1 -5844.38,E2 -5844.38} C_VEL
LIN {X 0,Y 502.191,Z 1085.149,A -85,B 0,C 180,E1 -5845.585,E2 -5845.585} C_VEL
LIN {X 0,Y 502.176,Z 1087.786,A -85,B 0,C 180,E1 -5846.389,E2 -5846.389} C_VEL
LIN {X 0,Y 502.093,Z 1090.68,A -85,B 0,C 180,E1 -5847.593,E2 -5847.593} C_VEL
LIN {X 0,Y 502.035,Z 1091.928,A -85,B 0,C 180,E1 -5848.395,E2 -5848.395} C_VEL
LIN {X 0,Y 501.987,Z 1092.706,A -85,B 0,C 180,E1 -5849.198,E2 -5849.198} C_VEL
LIN {X 0,Y 501.977,Z 1093,A -85,B 0,C 180,E1 -5850,E2 -5850} C_VEL
LIN {X 0,Y 501.987,Z 1092.706,A -85,B 0,C 180,E1 -5850.802,E2 -5850.802} C_VEL
LIN {X 0,Y 502.035,Z 1091.928,A -85,B 0,C 180,E1 -5851.604,E2 -5851.604} C_VEL
LIN {X 0,Y 502.093,Z 1090.679,A -85,B 0,C 180,E1 -5852.407,E2 -5852.407} C_VEL
LIN {X 0,Y 502.172,Z 1087.786,A -85,B 0,C 180,E1 -5853.611,E2 -5853.611} C_VEL
LIN {X 0,Y 502.193,Z 1085.149,A -85,B 0,C 180,E1 -5854.414,E2 -5854.414} C_VEL
LIN {X 0,Y 502.33,Z 1079.986,A -85,B 0,C 180,E1 -5855.62,E2 -5855.62} C_VEL
LIN {X 0,Y 502.43,Z 1073.932,A -85,B 0,C 180,E1 -5856.712,E2 -5856.712} C_VEL
LIN {X 0,Y 502.558,Z 1067.436,A -85,B 0,C 180,E1 -5857.634,E2 -5857.634} C_VEL
LIN {X 0,Y 502.818,Z 1059.407,A -85,B 0,C 180,E1 -5858.54,E2 -5858.54} C_VEL
LIN {X 0,Y 503.04,Z 1051.704,A -85,B 0,C 180,E1 -5859.245,E2 -5859.245} C_VEL
LIN {X 0,Y 503.232,Z 1043.597,A -85,B 0,C 180,E1 -5859.851,E2 -5859.851} C_VEL
LIN {X 0,Y 503.407,Z 1035.188,A -85,B 0,C 180,E1 -5860.355,E2 -5860.355} C_VEL
LIN {X 0,Y 503.592,Z 1026.597,A -85,B 0,C 180,E1 -5860.758,E2 -5860.758} C_VEL
LIN {X 0,Y 503.75,Z 1017.171,A -85,B 0,C 180,E1 -5861.085,E2 -5861.085} C_VEL
LIN {X 0,Y 503.961,Z 1006.384,A -85,B 0,C 180,E1 -5861.326,E2 -5861.326} C_VEL
LIN {X 0,Y 503.995,Z 941.597,A -85,B 0,C 180,E1 -5862.253,E2 -5862.253} C_VEL
LIN {X 0,Y 502.755,Z 932.478,A -85,B 0,C 180,E1 -5862.421,E2 -5862.421} C_VEL
LIN {X 0,Y 503.117,Z 915.734,A -85,B 0,C 180,E1 -5865.452,E2 -5865.452} C_VEL
LIN {X 0,Y 503.584,Z 897.877,A -85,B 0,C 180,E1 -5868.723,E2 -5868.723} C_VEL
LIN {X 0,Y 504.012,Z 881.938,A -85,B 0,C 180,E1 -5871.686,E2 -5871.686} C_VEL
LIN {X 0,Y 503.752,Z 877.772,A -85,B 0,C 180,E1 -5872.48,E2 -5872.48} C_VEL
LIN {X 0,Y 502.819,Z 872.666,A -85,B 0,C 180,E1 -5873.53,E2 -5873.53} C_VEL
LIN {X 0,Y 502.754,Z 872.674,A -85,B 0,C 180,E1 -5876.572,E2 -5876.572} C_VEL
LIN {X 0,Y 502.75,Z 872.676,A -85,B 0,C 180,E1 -5879.293,E2 -5879.293} C_VEL
LIN {X 0,Y 502.755,Z 872.67,A -85,B 0,C 180,E1 -5882.087,E2 -5882.087} C_VEL
LIN {X 0,Y 502.779,Z 872.669,A -85,B 0,C 180,E1 -5884.967,E2 -5884.967} C_VEL
LIN {X 0,Y 502.743,Z 872.67,A -85,B 0,C 180,E1 -5888.479,E2 -5888.479} C_VEL
LIN {X 0,Y 502.747,Z 872.669,A -85,B 0,C 180,E1 -5891.073,E2 -5891.073} C_VEL
LIN {X 0,Y 502.775,Z 872.666,A -85,B 0,C 180,E1 -5894.529,E2 -5894.529} C_VEL
LIN {X 0,Y 502.731,Z 872.677,A -85,B 0,C 180,E1 -5897.854,E2 -5897.854} C_VEL
LIN {X 0,Y 502.761,Z 872.667,A -85,B 0,C 180,E1 -5901.02,E2 -5901.02} C_VEL
LIN {X 0,Y 502.746,Z 872.675,A -85,B 0,C 180,E1 -5904.174,E2 -5904.174} C_VEL
LIN {X 0,Y 502.797,Z 872.665,A -85,B 0,C 180,E1 -5907,E2 -5907} C_VEL
LIN {X 0,Y 502.742,Z 872.672,A -85,B 0,C 180,E1 -5910.08,E2 -5910.08} C_VEL
LIN {X 0,Y 502.766,Z 872.674,A -85,B 0,C 180,E1 -5912.53,E2 -5912.53} C_VEL
LIN {X 0,Y 502.757,Z 872.673,A -85,B 0,C 180,E1 -5915.317,E2 -5915.317} C_VEL
LIN {X 0,Y 502.77,Z 872.669,A -85,B 0,C 180,E1 -5917.826,E2 -5917.826} C_VEL
LIN {X 0,Y 502.774,Z 872.669,A -85,B 0,C 180,E1 -5920.398,E2 -5920.398} C_VEL
LIN {X 0,Y 502.848,Z 872.852,A -85,B 0,C 180,E1 -5922.002,E2 -5922.002} C_VEL
LIN {X 0,Y 502.948,Z 878.134,A -85,B 0,C 180,E1 -5923.354,E2 -5923.354} C_VEL
LIN {X 0,Y 502.694,Z 889.56,A -85,B 0,C 180,E1 -5926.251,E2 -5926.251} C_VEL
LIN {X 0,Y 502.606,Z 895.255,A -85,B 0,C 180,E1 -5927.655,E2 -5927.655} C_VEL
LIN {X 0,Y 504.157,Z 906.085,A -85,B 0,C 180,E1 -5927.856,E2 -5927.856} C_VEL
LIN {X 0,Y 503.838,Z 970.195,A -85,B 0,C 180,E1 -5928.79,E2 -5928.79} C_VEL
LIN {X 0,Y 503.729,Z 980.024,A -85,B 0,C 180,E1 -5929.042,E2 -5929.042} C_VEL
LIN {X 0,Y 503.46,Z 991.661,A -85,B 0,C 180,E1 -5929.494,E2 -5929.494} C_VEL
LIN {X 0,Y 503.264,Z 1003.147,A -85,B 0,C 180,E1 -5930.15,E2 -5930.15} C_VEL
LIN {X 0,Y 503.042,Z 1012.563,A -85,B 0,C 180,E1 -5930.856,E2 -5930.856} C_VEL
LIN {X 0,Y 502.724,Z 1022.015,A -85,B 0,C 180,E1 -5931.762,E2 -5931.762} C_VEL
LIN {X 0,Y 502.549,Z 1030.18,A -85,B 0,C 180,E1 -5932.77,E2 -5932.77} C_VEL
LIN {X 0,Y 502.413,Z 1036.603,A -85,B 0,C 180,E1 -5933.777,E2 -5933.777} C_VEL
LIN {X 0,Y 502.218,Z 1041.782,A -85,B 0,C 180,E1 -5934.781,E2 -5934.781} C_VEL
LIN {X 0,Y 502.203,Z 1046.442,A -85,B 0,C 180,E1 -5935.988,E2 -5935.988} C_VEL
LIN {X 0,Y 502.135,Z 1048.819,A -85,B 0,C 180,E1 -5936.791,E2 -5936.791} C_VEL
LIN {X 0,Y 502.094,Z 1050.642,A -85,B 0,C 180,E1 -5937.594,E2 -5937.594} C_VEL
LIN {X 0,Y 502.035,Z 1051.936,A -85,B 0,C 180,E1 -5938.396,E2 -5938.396} C_VEL
LIN {X 0,Y 501.987,Z 1052.717,A -85,B 0,C 180,E1 -5939.198,E2 -5939.198} C_VEL
LIN {X 0,Y 501.978,Z 1052.997,A -85,B 0,C 180,E1 -5940,E2 -5940} C_VEL
LIN {X 0,Y 501.988,Z 1052.777,A -85,B 0,C 180,E1 -5940.803,E2 -5940.803} C_VEL
LIN {X 0,Y 502.036,Z 1052.058,A -85,B 0,C 180,E1 -5941.605,E2 -5941.605} C_VEL
LIN {X 0,Y 502.094,Z 1050.829,A -85,B 0,C 180,E1 -5942.407,E2 -5942.407} C_VEL
LIN {X 0,Y 502.17,Z 1047.956,A -85,B 0,C 180,E1 -5943.611,E2 -5943.611} C_VEL
LIN {X 0,Y 502.147,Z 1043.836,A -85,B 0,C 180,E1 -5944.818,E2 -5944.818} C_VEL
LIN {X 0,Y 502.428,Z 1038.25,A -85,B 0,C 180,E1 -5946.022,E2 -5946.022} C_VEL
LIN {X 0,Y 502.449,Z 1032.559,A -85,B 0,C 180,E1 -5946.971,E2 -5946.971} C_VEL
LIN {X 0,Y 502.67,Z 1024.517,A -85,B 0,C 180,E1 -5948.037,E2 -5948.037} C_VEL
LIN {X 0,Y 502.917,Z 1015.861,A -85,B 0,C 180,E1 -5948.944,E2 -5948.944} C_VEL
LIN {X 0,Y 503.218,Z 1005.967,A -85,B 0,C 180,E1 -5949.75,E2 -5949.75} C_VEL
LIN {X 0,Y 503.42,Z 996.191,A -85,B 0,C 180,E1 -5950.355,E2 -5950.355} C_VEL
LIN {X 0,Y 503.56,Z 987.853,A -85,B 0,C 180,E1 -5950.759,E2 -5950.759} C_VEL
LIN {X 0,Y 503.747,Z 978.825,A -85,B 0,C 180,E1 -5951.086,E2 -5951.086} C_VEL
LIN {X 0,Y 503.891,Z 970.063,A -85,B 0,C 180,E1 -5951.304,E2 -5951.304} C_VEL
LIN {X 0,Y 504.025,Z 904.594,A -85,B 0,C 180,E1 -5952.26,E2 -5952.26} C_VEL
LIN {X 0,Y 502.54,Z 894.957,A -85,B 0,C 180,E1 -5952.451,E2 -5952.451} C_VEL
LIN {X 0,Y 502.801,Z 883.077,A -85,B 0,C 180,E1 -5955.402,E2 -5955.402} C_VEL
LIN {X 0,Y 502.953,Z 873.097,A -85,B 0,C 180,E1 -5957.904,E2 -5957.904} C_VEL
LIN {X 0,Y 502.856,Z 872.661,A -85,B 0,C 180,E1 -5958.073,E2 -5958.073} C_VEL
LIN {X 0,Y 502.765,Z 872.671,A -85,B 0,C 180,E1 -5961.312,E2 -5961.312} C_VEL
LIN {X 0,Y 502.752,Z 872.668,A -85,B 0,C 180,E1 -5963.916,E2 -5963.916} C_VEL
LIN {X 0,Y 502.759,Z 872.667,A -85,B 0,C 180,E1 -5966.573,E2 -5966.573} C_VEL
LIN {X 0,Y 502.754,Z 872.674,A -85,B 0,C 180,E1 -5969.293,E2 -5969.293} C_VEL
LIN {X 0,Y 502.759,Z 872.669,A -85,B 0,C 180,E1 -5972.087,E2 -5972.087} C_VEL
LIN {X 0,Y 502.784,Z 872.664,A -85,B 0,C 180,E1 -5974.968,E2 -5974.968} C_VEL
LIN {X 0,Y 502.755,Z 872.668,A -85,B 0,C 180,E1 -5978.48,E2 -5978.48} C_VEL
LIN {X 0,Y 502.751,Z 872.667,A -85,B 0,C 180,E1 -5981.073,E2 -5981.073} C_VEL
LIN {X 0,Y 502.78,Z 872.667,A -85,B 0,C 180,E1 -5984.529,E2 -5984.529} C_VEL
LIN {X 0,Y 502.739,Z 872.672,A -85,B 0,C 180,E1 -5986.593,E2 -5986.593} C_VEL
LIN {X 0,Y 502.096,Z 872.757,A -85,B 0,C 180,E1 -5987.262,E2 -5987.262} C_VEL
LIN {X 0,Y 499.248,Z 873.112,A -85,B 0,C 180,E1 -5988.348,E2 -5988.348} C_VEL
LIN {X 0,Y 496.826,Z 873.408,A -85,B 0,C 180,E1 -5989.223,E2 -5989.223} C_VEL
LIN {X 0,Y 495.788,Z 873.538,A -85,B 0,C 180,E1 -5989.899,E2 -5989.899} C_VEL
LIN {X 0,Y 495.706,Z 873.55,A -85,B 0,C 180,E1 -5990.128,E2 -5990.128} C_VEL
LIN {X 0,Y 495.694,Z 873.554,A -85,B 0,C 180,E1 -5992.559,E2 -5992.559} C_VEL
LIN {X 0,Y 495.767,Z 873.538,A -85,B 0,C 180,E1 -5995.456,E2 -5995.456} C_VEL
LIN {X 0,Y 495.732,Z 873.545,A -85,B 0,C 180,E1 -5998.362,E2 -5998.362} C_VEL
LIN {X 0,Y 495.728,Z 873.543,A -85,B 0,C 180,E1 -6001.521,E2 -6001.521} C_VEL
LIN {X 0,Y 495.708,Z 873.545,A -85,B 0,C 180,E1 -6003.928,E2 -6003.928} C_VEL
LIN {X 0,Y 495.749,Z 873.548,A -85,B 0,C 180,E1 -6007.144,E2 -6007.144} C_VEL
LIN {X 0,Y 495.729,Z 873.542,A -85,B 0,C 180,E1 -6010.108,E2 -6010.108} C_VEL
LIN {X 0,Y 495.738,Z 873.542,A -85,B 0,C 180,E1 -6012.68,E2 -6012.68} C_VEL
LIN {X 0,Y 495.78,Z 873.541,A -85,B 0,C 180,E1 -6015.217,E2 -6015.217} C_VEL
LIN {X 0,Y 495.794,Z 873.534,A -85,B 0,C 180,E1 -6018.554,E2 -6018.554} C_VEL
LIN {X 0,Y 495.814,Z 873.539,A -85,B 0,C 180,E1 -6021.851,E2 -6021.851} C_VEL
LIN {X 0,Y 495.853,Z 873.53,A -85,B 0,C 180,E1 -6024.306,E2 -6024.306} C_VEL
LIN {X 0,Y 495.971,Z 873.515,A -85,B 0,C 180,E1 -6027.564,E2 -6027.564} C_VEL
LIN {X 0,Y 495.975,Z 873.519,A -85,B 0,C 180,E1 -6030,E2 -6030} C_VEL
LIN {X 0,Y 495.969,Z 873.518,A -85,B 0,C 180,E1 -6032.437,E2 -6032.437} C_VEL
LIN {X 0,Y 495.852,Z 873.527,A -85,B 0,C 180,E1 -6035.694,E2 -6035.694} C_VEL
LIN {X 0,Y 495.814,Z 873.535,A -85,B 0,C 180,E1 -6038.149,E2 -6038.149} C_VEL
LIN {X 0,Y 495.794,Z 873.534,A -85,B 0,C 180,E1 -6041.447,E2 -6041.447} C_VEL
LIN {X 0,Y 495.749,Z 873.549,A -85,B 0,C 180,E1 -6044.784,E2 -6044.784} C_VEL
LIN {X 0,Y 495.738,Z 873.544,A -85,B 0,C 180,E1 -6047.321,E2 -6047.321} C_VEL
LIN {X 0,Y 495.726,Z 873.542,A -85,B 0,C 180,E1 -6049.892,E2 -6049.892} C_VEL
LIN {X 0,Y 495.747,Z 873.545,A -85,B 0,C 180,E1 -6052.855,E2 -6052.855} C_VEL
LIN {X 0,Y 495.709,Z 873.545,A -85,B 0,C 180,E1 -6056.073,E2 -6056.073} C_VEL
LIN {X 0,Y 495.7,Z 873.547,A -85,B 0,C 180,E1 -6058.82,E2 -6058.82} C_VEL
LIN {X 0,Y 495.729,Z 873.548,A -85,B 0,C 180,E1 -6061.719,E2 -6061.719} C_VEL
LIN {X 0,Y 495.742,Z 873.54,A -85,B 0,C 180,E1 -6064.688,E2 -6064.688} C_VEL
LIN {X 0,Y 495.693,Z 873.552,A -85,B 0,C 180,E1 -6067.565,E2 -6067.565} C_VEL
LIN {X 0,Y 495.71,Z 873.551,A -85,B 0,C 180,E1 -6070.039,E2 -6070.039} C_VEL
LIN {X 0,Y 495.693,Z 873.547,A -85,B 0,C 180,E1 -6072.887,E2 -6072.887} C_VEL
LIN {X 0,Y 495.717,Z 873.55,A -85,B 0,C 180,E1 -6075.996,E2 -6075.996} C_VEL
LIN {X 0,Y 495.712,Z 873.544,A -85,B 0,C 180,E1 -6079.294,E2 -6079.294} C_VEL
LIN {X 0,Y 495.71,Z 873.544,A -85,B 0,C 180,E1 -6081.404,E2 -6081.404} C_VEL
LIN {X 0,Y 495.73,Z 873.55,A -85,B 0,C 180,E1 -6084.46,E2 -6084.46} C_VEL
LIN {X 0,Y 495.744,Z 873.541,A -85,B 0,C 180,E1 -6087.403,E2 -6087.403} C_VEL
LIN {X 0,Y 495.699,Z 873.548,A -85,B 0,C 180,E1 -6090.249,E2 -6090.249} C_VEL
LIN {X 0,Y 495.724,Z 873.547,A -85,B 0,C 180,E1 -6093.275,E2 -6093.275} C_VEL
LIN {X 0,Y 495.705,Z 873.546,A -85,B 0,C 180,E1 -6095.722,E2 -6095.722} C_VEL
LIN {X 0,Y 495.735,Z 873.542,A -85,B 0,C 180,E1 -6098.37,E2 -6098.37} C_VEL
LIN {X 0,Y 495.755,Z 873.543,A -85,B 0,C 180,E1 -6100.97,E2 -6100.97} C_VEL
LIN {X 0,Y 495.746,Z 873.547,A -85,B 0,C 180,E1 -6103.528,E2 -6103.528} C_VEL
LIN {X 0,Y 495.764,Z 873.54,A -85,B 0,C 180,E1 -6106.054,E2 -6106.054} C_VEL
LIN {X 0,Y 495.792,Z 873.534,A -85,B 0,C 180,E1 -6108.553,E2 -6108.553} C_VEL
LIN {X 0,Y 495.812,Z 873.539,A -85,B 0,C 180,E1 -6111.851,E2 -6111.851} C_VEL
LIN {X 0,Y 495.851,Z 873.53,A -85,B 0,C 180,E1 -6114.306,E2 -6114.306} C_VEL
LIN {X 0,Y 495.969,Z 873.515,A -85,B 0,C 180,E1 -6117.563,E2 -6117.563} C_VEL
LIN {X 0,Y 495.973,Z 873.519,A -85,B 0,C 180,E1 -6120,E2 -6120} C_VEL
LIN {X 0,Y 495.967,Z 873.518,A -85,B 0,C 180,E1 -6122.436,E2 -6122.436} C_VEL
LIN {X 0,Y 495.85,Z 873.528,A -85,B 0,C 180,E1 -6125.694,E2 -6125.694} C_VEL
LIN {X 0,Y 495.811,Z 873.536,A -85,B 0,C 180,E1 -6128.149,E2 -6128.149} C_VEL
LIN {X 0,Y 495.791,Z 873.534,A -85,B 0,C 180,E1 -6131.446,E2 -6131.446} C_VEL
LIN {X 0,Y 495.765,Z 873.546,A -85,B 0,C 180,E1 -6134.783,E2 -6134.783} C_VEL
LIN {X 0,Y 495.763,Z 873.538,A -85,B 0,C 180,E1 -6138.172,E2 -6138.172} C_VEL
LIN {X 0,Y 495.765,Z 873.542,A -85,B 0,C 180,E1 -6140.756,E2 -6140.756} C_VEL
LIN {X 0,Y 495.725,Z 873.548,A -85,B 0,C 180,E1 -6143.388,E2 -6143.388} C_VEL
LIN {X 0,Y 495.705,Z 873.545,A -85,B 0,C 180,E1 -6146.072,E2 -6146.072} C_VEL
LIN {X 0,Y 495.696,Z 873.548,A -85,B 0,C 180,E1 -6148.819,E2 -6148.819} C_VEL
LIN {X 0,Y 495.725,Z 873.548,A -85,B 0,C 180,E1 -6151.719,E2 -6151.719} C_VEL
LIN {X 0,Y 495.738,Z 873.541,A -85,B 0,C 180,E1 -6154.688,E2 -6154.688} C_VEL
LIN {X 0,Y 495.689,Z 873.553,A -85,B 0,C 180,E1 -6157.565,E2 -6157.565} C_VEL
LIN {X 0,Y 495.706,Z 873.551,A -85,B 0,C 180,E1 -6160.039,E2 -6160.039} C_VEL
LIN {X 0,Y 495.689,Z 873.547,A -85,B 0,C 180,E1 -6162.887,E2 -6162.887} C_VEL
LIN {X 0,Y 495.712,Z 873.551,A -85,B 0,C 180,E1 -6165.996,E2 -6165.996} C_VEL
LIN {X 0,Y 495.707,Z 873.544,A -85,B 0,C 180,E1 -6169.294,E2 -6169.294} C_VEL
LIN {X 0,Y 495.706,Z 873.545,A -85,B 0,C 180,E1 -6171.404,E2 -6171.404} C_VEL
LIN {X 0,Y 495.726,Z 873.551,A -85,B 0,C 180,E1 -6174.46,E2 -6174.46} C_VEL
LIN {X 0,Y 495.739,Z 873.541,A -85,B 0,C 180,E1 -6177.403,E2 -6177.403} C_VEL
LIN {X 0,Y 495.694,Z 873.548,A -85,B 0,C 180,E1 -6180.249,E2 -6180.249} C_VEL
LIN {X 0,Y 495.719,Z 873.552,A -85,B 0,C 180,E1 -6183.275,E2 -6183.275} C_VEL
LIN {X 0,Y 495.777,Z 873.679,A -85,B 0,C 180,E1 -6186.254,E2 -6186.254} C_VEL
LIN {X 0,Y 497.092,Z 881.182,A -85,B 0,C 180,E1 -6187.778,E2 -6187.778} C_VEL
LIN {X 0,Y 496.739,Z 894.748,A -85,B 0,C 180,E1 -6190.365,E2 -6190.365} C_VEL
LIN {X 0,Y 496.277,Z 910.536,A -85,B 0,C 180,E1 -6193.335,E2 -6193.335} C_VEL
LIN {X 0,Y 495.824,Z 927.412,A -85,B 0,C 180,E1 -6196.474,E2 -6196.474} C_VEL
LIN {X 0,Y 495.739,Z 932.745,A -85,B 0,C 180,E1 -6197.422,E2 -6197.422} C_VEL
LIN {X 0,Y 497.157,Z 943.72,A -85,B 0,C 180,E1 -6197.615,E2 -6197.615} C_VEL
LIN {X 0,Y 496.96,Z 1007.859,A -85,B 0,C 180,E1 -6198.559,E2 -6198.559} C_VEL
LIN {X 0,Y 496.74,Z 1017.31,A -85,B 0,C 180,E1 -6198.782,E2 -6198.782} C_VEL
LIN {X 0,Y 496.622,Z 1026,A -85,B 0,C 180,E1 -6199.089,E2 -6199.089} C_VEL
LIN {X 0,Y 496.396,Z 1034.65,A -85,B 0,C 180,E1 -6199.497,E2 -6199.497} C_VEL
LIN {X 0,Y 496.224,Z 1043.103,A -85,B 0,C 180,E1 -6200.009,E2 -6200.009} C_VEL
LIN {X 0,Y 496.002,Z 1051.239,A -85,B 0,C 180,E1 -6200.622,E2 -6200.622} C_VEL
LIN {X 0,Y 495.771,Z 1058.976,A -85,B 0,C 180,E1 -6201.337,E2 -6201.337} C_VEL
LIN {X 0,Y 495.525,Z 1067.087,A -85,B 0,C 180,E1 -6202.256,E2 -6202.256} C_VEL
LIN {X 0,Y 495.358,Z 1074.203,A -85,B 0,C 180,E1 -6203.284,E2 -6203.284} C_VEL
LIN {X 0,Y 495.255,Z 1079.777,A -85,B 0,C 180,E1 -6204.299,E2 -6204.299} C_VEL
LIN {X 0,Y 495.085,Z 1084.982,A -85,B 0,C 180,E1 -6205.522,E2 -6205.522} C_VEL
LIN {X 0,Y 495.1,Z 1087.648,A -85,B 0,C 180,E1 -6206.337,E2 -6206.337} C_VEL
LIN {X 0,Y 495,Z 1090.565,A -85,B 0,C 180,E1 -6207.559,E2 -6207.559} C_VEL
LIN {X 0,Y 494.961,Z 1091.824,A -85,B 0,C 180,E1 -6208.373,E2 -6208.373} C_VEL
LIN {X 0,Y 494.907,Z 1092.607,A -85,B 0,C 180,E1 -6209.186,E2 -6209.186} C_VEL
LIN {X 0,Y 494.895,Z 1092.902,A -85,B 0,C 180,E1 -6210,E2 -6210} C_VEL
LIN {X 0,Y 494.907,Z 1092.606,A -85,B 0,C 180,E1 -6210.814,E2 -6210.814} C_VEL
LIN {X 0,Y 494.961,Z 1091.822,A -85,B 0,C 180,E1 -6211.627,E2 -6211.627} C_VEL
LIN {X 0,Y 495,Z 1090.562,A -85,B 0,C 180,E1 -6212.441,E2 -6212.441} C_VEL
LIN {X 0,Y 495.097,Z 1087.643,A -85,B 0,C 180,E1 -6213.662,E2 -6213.662} C_VEL
LIN {X 0,Y 495.087,Z 1084.974,A -85,B 0,C 180,E1 -6214.478,E2 -6214.478} C_VEL
LIN {X 0,Y 495.256,Z 1079.761,A -85,B 0,C 180,E1 -6215.701,E2 -6215.701} C_VEL
LIN {X 0,Y 495.378,Z 1073.139,A -85,B 0,C 180,E1 -6216.885,E2 -6216.885} C_VEL
LIN {X 0,Y 495.553,Z 1065.331,A -85,B 0,C 180,E1 -6217.948,E2 -6217.948} C_VEL
LIN {X 0,Y 495.806,Z 1057.898,A -85,B 0,C 180,E1 -6218.765,E2 -6218.765} C_VEL
LIN {X 0,Y 496.042,Z 1049.926,A -85,B 0,C 180,E1 -6219.48,E2 -6219.48} C_VEL
LIN {X 0,Y 496.358,Z 1039.972,A -85,B 0,C 180,E1 -6220.194,E2 -6220.194} C_VEL
LIN {X 0,Y 496.52,Z 1029.456,A -85,B 0,C 180,E1 -6220.758,E2 -6220.758} C_VEL
LIN {X 0,Y 496.709,Z 1018.715,A -85,B 0,C 180,E1 -6221.167,E2 -6221.167} C_VEL
LIN {X 0,Y 496.915,Z 1009.851,A -85,B 0,C 180,E1 -6221.394,E2 -6221.394} C_VEL
LIN {X 0,Y 497.075,Z 967.935,A -85,B 0,C 180,E1 -6222.031,E2 -6222.031} C_VEL
LIN {X 0,Y 497.116,Z 942.785,A -85,B 0,C 180,E1 -6222.393,E2 -6222.393} C_VEL
LIN {X 0,Y 495.716,Z 932.18,A -85,B 0,C 180,E1 -6222.593,E2 -6222.593} C_VEL
LIN {X 0,Y 496.084,Z 915.732,A -85,B 0,C 180,E1 -6225.615,E2 -6225.615} C_VEL
LIN {X 0,Y 496.538,Z 899.225,A -85,B 0,C 180,E1 -6228.682,E2 -6228.682} C_VEL
LIN {X 0,Y 497.035,Z 882.758,A -85,B 0,C 180,E1 -6231.788,E2 -6231.788} C_VEL
LIN {X 0,Y 496.551,Z 877.987,A -85,B 0,C 180,E1 -6232.728,E2 -6232.728} C_VEL
LIN {X 0,Y 495.755,Z 873.545,A -85,B 0,C 180,E1 -6233.664,E2 -6233.664} C_VEL
LIN {X 0,Y 495.715,Z 873.554,A -85,B 0,C 180,E1 -6236.98,E2 -6236.98} C_VEL
LIN {X 0,Y 495.693,Z 873.551,A -85,B 0,C 180,E1 -6239.751,E2 -6239.751} C_VEL
LIN {X 0,Y 495.738,Z 873.544,A -85,B 0,C 180,E1 -6242.597,E2 -6242.597} C_VEL
LIN {X 0,Y 495.724,Z 873.552,A -85,B 0,C 180,E1 -6245.54,E2 -6245.54} C_VEL
LIN {X 0,Y 495.72,Z 873.545,A -85,B 0,C 180,E1 -6248.762,E2 -6248.762} C_VEL
LIN {X 0,Y 495.697,Z 873.554,A -85,B 0,C 180,E1 -6251.787,E2 -6251.787} C_VEL
LIN {X 0,Y 495.729,Z 873.544,A -85,B 0,C 180,E1 -6255.142,E2 -6255.142} C_VEL
LIN {X 0,Y 495.697,Z 873.553,A -85,B 0,C 180,E1 -6258.213,E2 -6258.213} C_VEL
LIN {X 0,Y 495.705,Z 873.547,A -85,B 0,C 180,E1 -6261.404,E2 -6261.404} C_VEL
LIN {X 0,Y 495.724,Z 873.55,A -85,B 0,C 180,E1 -6264.461,E2 -6264.461} C_VEL
LIN {X 0,Y 495.738,Z 873.542,A -85,B 0,C 180,E1 -6267.404,E2 -6267.404} C_VEL
LIN {X 0,Y 495.693,Z 873.552,A -85,B 0,C 180,E1 -6270.249,E2 -6270.249} C_VEL
LIN {X 0,Y 495.719,Z 873.547,A -85,B 0,C 180,E1 -6273.275,E2 -6273.275} C_VEL
LIN {X 0,Y 495.69,Z 873.551,A -85,B 0,C 180,E1 -6275.722,E2 -6275.722} C_VEL
LIN {X 0,Y 495.727,Z 873.549,A -85,B 0,C 180,E1 -6278.371,E2 -6278.371} C_VEL
LIN {X 0,Y 495.75,Z 873.549,A -85,B 0,C 180,E1 -6280.971,E2 -6280.971} C_VEL
LIN {X 0,Y 495.795,Z 873.704,A -85,B 0,C 180,E1 -6281.883,E2 -6281.883} C_VEL
LIN {X 0,Y 495.978,Z 878.429,A -85,B 0,C 180,E1 -6283.113,E2 -6283.113} C_VEL
LIN {X 0,Y 495.685,Z 889.885,A -85,B 0,C 180,E1 -6286.053,E2 -6286.053} C_VEL
LIN {X 0,Y 495.574,Z 895.476,A -85,B 0,C 180,E1 -6287.474,E2 -6287.474} C_VEL
LIN {X 0,Y 497.217,Z 907.154,A -85,B 0,C 180,E1 -6287.702,E2 -6287.702} C_VEL
LIN {X 0,Y 496.853,Z 970.885,A -85,B 0,C 180,E1 -6288.656,E2 -6288.656} C_VEL
LIN {X 0,Y 496.726,Z 981.378,A -85,B 0,C 180,E1 -6288.937,E2 -6288.937} C_VEL
LIN {X 0,Y 496.449,Z 992.601,A -85,B 0,C 180,E1 -6289.395,E2 -6289.395} C_VEL
LIN {X 0,Y 496.257,Z 1003.173,A -85,B 0,C 180,E1 -6290.01,E2 -6290.01} C_VEL
LIN {X 0,Y 496.032,Z 1012.668,A -85,B 0,C 180,E1 -6290.726,E2 -6290.726} C_VEL
LIN {X 0,Y 495.7,Z 1022.168,A -85,B 0,C 180,E1 -6291.644,E2 -6291.644} C_VEL
LIN {X 0,Y 495.498,Z 1030.362,A -85,B 0,C 180,E1 -6292.666,E2 -6292.666} C_VEL
LIN {X 0,Y 495.353,Z 1036.826,A -85,B 0,C 180,E1 -6293.688,E2 -6293.688} C_VEL
LIN {X 0,Y 495.159,Z 1042.01,A -85,B 0,C 180,E1 -6294.707,E2 -6294.707} C_VEL
LIN {X 0,Y 495.143,Z 1046.712,A -85,B 0,C 180,E1 -6295.931,E2 -6295.931} C_VEL
LIN {X 0,Y 495.06,Z 1049.084,A -85,B 0,C 180,E1 -6296.745,E2 -6296.745} C_VEL
LIN {X 0,Y 495.014,Z 1050.895,A -85,B 0,C 180,E1 -6297.559,E2 -6297.559} C_VEL
LIN {X 0,Y 494.961,Z 1052.192,A -85,B 0,C 180,E1 -6298.373,E2 -6298.373} C_VEL
LIN {X 0,Y 494.908,Z 1052.975,A -85,B 0,C 180,E1 -6299.187,E2 -6299.187} C_VEL
LIN {X 0,Y 494.896,Z 1053.25,A -85,B 0,C 180,E1 -6300,E2 -6300} C_VEL
LIN {X 0,Y 494.908,Z 1053.019,A -85,B 0,C 180,E1 -6300.814,E2 -6300.814} C_VEL
LIN {X 0,Y 494.962,Z 1052.291,A -85,B 0,C 180,E1 -6301.628,E2 -6301.628} C_VEL
LIN {X 0,Y 495.001,Z 1051.064,A -85,B 0,C 180,E1 -6302.442,E2 -6302.442} C_VEL
LIN {X 0,Y 495.095,Z 1048.207,A -85,B 0,C 180,E1 -6303.663,E2 -6303.663} C_VEL
LIN {X 0,Y 495.072,Z 1044.068,A -85,B 0,C 180,E1 -6304.887,E2 -6304.887} C_VEL
LIN {X 0,Y 495.364,Z 1038.445,A -85,B 0,C 180,E1 -6306.109,E2 -6306.109} C_VEL
LIN {X 0,Y 495.41,Z 1032.352,A -85,B 0,C 180,E1 -6307.131,E2 -6307.131} C_VEL
LIN {X 0,Y 495.629,Z 1024.645,A -85,B 0,C 180,E1 -6308.152,E2 -6308.152} C_VEL
LIN {X 0,Y 495.923,Z 1015.946,A -85,B 0,C 180,E1 -6309.071,E2 -6309.071} C_VEL
LIN {X 0,Y 496.222,Z 1005.987,A -85,B 0,C 180,E1 -6309.889,E2 -6309.889} C_VEL
LIN {X 0,Y 496.449,Z 996.14,A -85,B 0,C 180,E1 -6310.502,E2 -6310.502} C_VEL
LIN {X 0,Y 496.581,Z 987.716,A -85,B 0,C 180,E1 -6310.912,E2 -6310.912} C_VEL
LIN {X 0,Y 496.795,Z 978.554,A -85,B 0,C 180,E1 -6311.243,E2 -6311.243} C_VEL
LIN {X 0,Y 496.923,Z 968.558,A -85,B 0,C 180,E1 -6311.484,E2 -6311.484} C_VEL
LIN {X 0,Y 497.022,Z 904.722,A -85,B 0,C 180,E1 -6312.431,E2 -6312.431} C_VEL
LIN {X 0,Y 495.527,Z 895.2,A -85,B 0,C 180,E1 -6312.627,E2 -6312.627} C_VEL
LIN {X 0,Y 495.804,Z 883.27,A -85,B 0,C 180,E1 -6315.625,E2 -6315.625} C_VEL
LIN {X 0,Y 495.93,Z 874.064,A -85,B 0,C 180,E1 -6317.953,E2 -6317.953} C_VEL
LIN {X 0,Y 495.811,Z 873.539,A -85,B 0,C 180,E1 -6318.171,E2 -6318.171} C_VEL
LIN {X 0,Y 495.73,Z 873.544,A -85,B 0,C 180,E1 -6321.63,E2 -6321.63} C_VEL
LIN {X 0,Y 495.702,Z 873.545,A -85,B 0,C 180,E1 -6324.278,E2 -6324.278} C_VEL
LIN {X 0,Y 495.719,Z 873.547,A -85,B 0,C 180,E1 -6326.98,E2 -6326.98} C_VEL
LIN {X 0,Y 495.697,Z 873.551,A -85,B 0,C 180,E1 -6329.752,E2 -6329.752} C_VEL
LIN {X 0,Y 495.742,Z 873.54,A -85,B 0,C 180,E1 -6332.597,E2 -6332.597} C_VEL
LIN {X 0,Y 495.729,Z 873.549,A -85,B 0,C 180,E1 -6335.54,E2 -6335.54} C_VEL
LIN {X 0,Y 495.73,Z 873.542,A -85,B 0,C 180,E1 -6338.763,E2 -6338.763} C_VEL
LIN {X 0,Y 495.703,Z 873.551,A -85,B 0,C 180,E1 -6341.787,E2 -6341.787} C_VEL
LIN {X 0,Y 495.733,Z 873.541,A -85,B 0,C 180,E1 -6345.142,E2 -6345.142} C_VEL
LIN {X 0,Y 495.702,Z 873.554,A -85,B 0,C 180,E1 -6348.213,E2 -6348.213} C_VEL
LIN {X 0,Y 495.706,Z 873.55,A -85,B 0,C 180,E1 -6350.128,E2 -6350.128} C_VEL
LIN {X 0,Y 495.044,Z 873.639,A -85,B 0,C 180,E1 -6350.806,E2 -6350.806} C_VEL
LIN {X 0,Y 492.19,Z 873.992,A -85,B 0,C 180,E1 -6351.907,E2 -6351.907} C_VEL
LIN {X 0,Y 489.772,Z 874.288,A -85,B 0,C 180,E1 -6352.795,E2 -6352.795} C_VEL
LIN {X 0,Y 488.732,Z 874.414,A -85,B 0,C 180,E1 -6353.48,E2 -6353.48} C_VEL
LIN {X 0,Y 488.647,Z 874.425,A -85,B 0,C 180,E1 -6353.712,E2 -6353.712} C_VEL
LIN {X 0,Y 488.711,Z 874.424,A -85,B 0,C 180,E1 -6356.521,E2 -6356.521} C_VEL
LIN {X 0,Y 488.666,Z 874.422,A -85,B 0,C 180,E1 -6359.777,E2 -6359.777} C_VEL
LIN {X 0,Y 488.678,Z 874.425,A -85,B 0,C 180,E1 -6362.599,E2 -6362.599} C_VEL
LIN {X 0,Y 488.692,Z 874.423,A -85,B 0,C 180,E1 -6365.351,E2 -6365.351} C_VEL
LIN {X 0,Y 488.691,Z 874.419,A -85,B 0,C 180,E1 -6368.043,E2 -6368.043} C_VEL
LIN {X 0,Y 488.714,Z 874.417,A -85,B 0,C 180,E1 -6370.686,E2 -6370.686} C_VEL
LIN {X 0,Y 488.758,Z 874.411,A -85,B 0,C 180,E1 -6374.145,E2 -6374.145} C_VEL
LIN {X 0,Y 488.735,Z 874.422,A -85,B 0,C 180,E1 -6377.544,E2 -6377.544} C_VEL
LIN {X 0,Y 488.728,Z 874.414,A -85,B 0,C 180,E1 -6380.899,E2 -6380.899} C_VEL
LIN {X 0,Y 488.778,Z 874.411,A -85,B 0,C 180,E1 -6383.395,E2 -6383.395} C_VEL
LIN {X 0,Y 488.658,Z 874.431,A -85,B 0,C 180,E1 -6385.876,E2 -6385.876} C_VEL
LIN {X 0,Y 488.936,Z 874.391,A -85,B 0,C 180,E1 -6387.529,E2 -6387.529} C_VEL
LIN {X 0,Y 488.944,Z 874.395,A -85,B 0,C 180,E1 -6390,E2 -6390} C_VEL
LIN {X 0,Y 488.935,Z 874.394,A -85,B 0,C 180,E1 -6392.472,E2 -6392.472} C_VEL
LIN {X 0,Y 488.813,Z 874.405,A -85,B 0,C 180,E1 -6395.776,E2 -6395.776} C_VEL
LIN {X 0,Y 488.758,Z 874.416,A -85,B 0,C 180,E1 -6398.268,E2 -6398.268} C_VEL
LIN {X 0,Y 488.763,Z 874.41,A -85,B 0,C 180,E1 -6401.614,E2 -6401.614} C_VEL
LIN {X 0,Y 488.719,Z 874.421,A -85,B 0,C 180,E1 -6405.002,E2 -6405.002} C_VEL
LIN {X 0,Y 488.711,Z 874.418,A -85,B 0,C 180,E1 -6408.353,E2 -6408.353} C_VEL
LIN {X 0,Y 488.704,Z 874.426,A -85,B 0,C 180,E1 -6411.071,E2 -6411.071} C_VEL
LIN {X 0,Y 488.658,Z 874.425,A -85,B 0,C 180,E1 -6413.748,E2 -6413.748} C_VEL
LIN {X 0,Y 488.671,Z 874.421,A -85,B 0,C 180,E1 -6416.477,E2 -6416.477} C_VEL
LIN {X 0,Y 488.663,Z 874.429,A -85,B 0,C 180,E1 -6419.275,E2 -6419.275} C_VEL
LIN {X 0,Y 488.679,Z 874.422,A -85,B 0,C 180,E1 -6422.149,E2 -6422.149} C_VEL
LIN {X 0,Y 488.699,Z 874.419,A -85,B 0,C 180,E1 -6425.117,E2 -6425.117} C_VEL
LIN {X 0,Y 488.647,Z 874.428,A -85,B 0,C 180,E1 -6428.203,E2 -6428.203} C_VEL
LIN {X 0,Y 488.647,Z 874.426,A -85,B 0,C 180,E1 -6431.422,E2 -6431.422} C_VEL
LIN {X 0,Y 488.7,Z 874.419,A -85,B 0,C 180,E1 -6434.803,E2 -6434.803} C_VEL
LIN {X 0,Y 488.651,Z 874.424,A -85,B 0,C 180,E1 -6437.469,E2 -6437.469} C_VEL
LIN {X 0,Y 488.669,Z 874.425,A -85,B 0,C 180,E1 -6440.742,E2 -6440.742} C_VEL
LIN {X 0,Y 488.643,Z 874.426,A -85,B 0,C 180,E1 -6443.864,E2 -6443.864} C_VEL
LIN {X 0,Y 488.712,Z 874.424,A -85,B 0,C 180,E1 -6446.521,E2 -6446.521} C_VEL
LIN {X 0,Y 488.667,Z 874.422,A -85,B 0,C 180,E1 -6449.776,E2 -6449.776} C_VEL
LIN {X 0,Y 488.678,Z 874.425,A -85,B 0,C 180,E1 -6452.599,E2 -6452.599} C_VEL
LIN {X 0,Y 488.692,Z 874.423,A -85,B 0,C 180,E1 -6455.351,E2 -6455.351} C_VEL
LIN {X 0,Y 488.69,Z 874.419,A -85,B 0,C 180,E1 -6458.042,E2 -6458.042} C_VEL
LIN {X 0,Y 488.714,Z 874.418,A -85,B 0,C 180,E1 -6460.685,E2 -6460.685} C_VEL
LIN {X 0,Y 488.696,Z 874.426,A -85,B 0,C 180,E1 -6463.284,E2 -6463.284} C_VEL
LIN {X 0,Y 488.71,Z 874.42,A -85,B 0,C 180,E1 -6465.849,E2 -6465.849} C_VEL
LIN {X 0,Y 488.761,Z 874.41,A -85,B 0,C 180,E1 -6468.386,E2 -6468.386} C_VEL
LIN {X 0,Y 488.756,Z 874.42,A -85,B 0,C 180,E1 -6471.732,E2 -6471.732} C_VEL
LIN {X 0,Y 488.811,Z 874.407,A -85,B 0,C 180,E1 -6474.223,E2 -6474.223} C_VEL
LIN {X 0,Y 488.934,Z 874.391,A -85,B 0,C 180,E1 -6477.528,E2 -6477.528} C_VEL
LIN {X 0,Y 488.942,Z 874.395,A -85,B 0,C 180,E1 -6480,E2 -6480} C_VEL
LIN {X 0,Y 488.933,Z 874.394,A -85,B 0,C 180,E1 -6482.471,E2 -6482.471} C_VEL
LIN {X 0,Y 488.81,Z 874.405,A -85,B 0,C 180,E1 -6485.776,E2 -6485.776} C_VEL
LIN {X 0,Y 488.755,Z 874.417,A -85,B 0,C 180,E1 -6488.267,E2 -6488.267} C_VEL
LIN {X 0,Y 488.76,Z 874.41,A -85,B 0,C 180,E1 -6491.613,E2 -6491.613} C_VEL
LIN {X 0,Y 488.727,Z 874.42,A -85,B 0,C 180,E1 -6495.001,E2 -6495.001} C_VEL
LIN {X 0,Y 488.707,Z 874.419,A -85,B 0,C 180,E1 -6498.444,E2 -6498.444} C_VEL
LIN {X 0,Y 488.7,Z 874.426,A -85,B 0,C 180,E1 -6501.071,E2 -6501.071} C_VEL
LIN {X 0,Y 488.654,Z 874.425,A -85,B 0,C 180,E1 -6503.747,E2 -6503.747} C_VEL
LIN {X 0,Y 488.668,Z 874.422,A -85,B 0,C 180,E1 -6506.477,E2 -6506.477} C_VEL
LIN {X 0,Y 488.659,Z 874.43,A -85,B 0,C 180,E1 -6509.274,E2 -6509.274} C_VEL
LIN {X 0,Y 488.675,Z 874.422,A -85,B 0,C 180,E1 -6512.149,E2 -6512.149} C_VEL
LIN {X 0,Y 488.695,Z 874.42,A -85,B 0,C 180,E1 -6515.117,E2 -6515.117} C_VEL
LIN {X 0,Y 488.643,Z 874.428,A -85,B 0,C 180,E1 -6518.203,E2 -6518.203} C_VEL
LIN {X 0,Y 488.642,Z 874.427,A -85,B 0,C 180,E1 -6521.422,E2 -6521.422} C_VEL
LIN {X 0,Y 488.695,Z 874.419,A -85,B 0,C 180,E1 -6524.803,E2 -6524.803} C_VEL
LIN {X 0,Y 488.647,Z 874.425,A -85,B 0,C 180,E1 -6527.469,E2 -6527.469} C_VEL
LIN {X 0,Y 488.665,Z 874.425,A -85,B 0,C 180,E1 -6530.742,E2 -6530.742} C_VEL
LIN {X 0,Y 488.639,Z 874.426,A -85,B 0,C 180,E1 -6533.864,E2 -6533.864} C_VEL
LIN {X 0,Y 488.707,Z 874.425,A -85,B 0,C 180,E1 -6536.521,E2 -6536.521} C_VEL
LIN {X 0,Y 488.662,Z 874.422,A -85,B 0,C 180,E1 -6539.776,E2 -6539.776} C_VEL
LIN {X 0,Y 488.673,Z 874.426,A -85,B 0,C 180,E1 -6542.599,E2 -6542.599} C_VEL
LIN {X 0,Y 488.712,Z 874.506,A -85,B 0,C 180,E1 -6546.086,E2 -6546.086} C_VEL
LIN {X 0,Y 490.161,Z 883.242,A -85,B 0,C 180,E1 -6547.89,E2 -6547.89} C_VEL
LIN {X 0,Y 489.718,Z 897.933,A -85,B 0,C 180,E1 -6550.726,E2 -6550.726} C_VEL
LIN {X 0,Y 489.15,Z 915.967,A -85,B 0,C 180,E1 -6554.158,E2 -6554.158} C_VEL
LIN {X 0,Y 488.664,Z 932.178,A -85,B 0,C 180,E1 -6557.222,E2 -6557.222} C_VEL
LIN {X 0,Y 490.222,Z 944.876,A -85,B 0,C 180,E1 -6557.466,E2 -6557.466} C_VEL
LIN {X 0,Y 490.004,Z 1006.919,A -85,B 0,C 180,E1 -6558.395,E2 -6558.395} C_VEL
LIN {X 0,Y 489.779,Z 1016.552,A -85,B 0,C 180,E1 -6558.62,E2 -6558.62} C_VEL
LIN {X 0,Y 489.616,Z 1026.579,A -85,B 0,C 180,E1 -6558.983,E2 -6558.983} C_VEL
LIN {X 0,Y 489.364,Z 1035.974,A -85,B 0,C 180,E1 -6559.449,E2 -6559.449} C_VEL
LIN {X 0,Y 489.139,Z 1045.616,A -85,B 0,C 180,E1 -6560.071,E2 -6560.071} C_VEL
LIN {X 0,Y 488.82,Z 1055.469,A -85,B 0,C 180,E1 -6560.9,E2 -6560.9} C_VEL
LIN {X 0,Y 488.579,Z 1063.26,A -85,B 0,C 180,E1 -6561.729,E2 -6561.729} C_VEL
LIN {X 0,Y 488.39,Z 1069.674,A -85,B 0,C 180,E1 -6562.558,E2 -6562.558} C_VEL
LIN {X 0,Y 488.267,Z 1075.003,A -85,B 0,C 180,E1 -6563.388,E2 -6563.388} C_VEL
LIN {X 0,Y 488.188,Z 1079.447,A -85,B 0,C 180,E1 -6564.216,E2 -6564.216} C_VEL
LIN {X 0,Y 487.989,Z 1084.667,A -85,B 0,C 180,E1 -6565.457,E2 -6565.457} C_VEL
LIN {X 0,Y 488.025,Z 1087.347,A -85,B 0,C 180,E1 -6566.284,E2 -6566.284} C_VEL
LIN {X 0,Y 487.911,Z 1090.273,A -85,B 0,C 180,E1 -6567.523,E2 -6567.523} C_VEL
LIN {X 0,Y 487.889,Z 1091.54,A -85,B 0,C 180,E1 -6568.349,E2 -6568.349} C_VEL
LIN {X 0,Y 487.83,Z 1092.325,A -85,B 0,C 180,E1 -6569.174,E2 -6569.174} C_VEL
LIN {X 0,Y 487.816,Z 1092.62,A -85,B 0,C 180,E1 -6570,E2 -6570} C_VEL
LIN {X 0,Y 487.83,Z 1092.322,A -85,B 0,C 180,E1 -6570.825,E2 -6570.825} C_VEL
LIN {X 0,Y 487.889,Z 1091.534,A -85,B 0,C 180,E1 -6571.651,E2 -6571.651} C_VEL
LIN {X 0,Y 487.911,Z 1090.262,A -85,B 0,C 180,E1 -6572.477,E2 -6572.477} C_VEL
LIN {X 0,Y 488.022,Z 1087.329,A -85,B 0,C 180,E1 -6573.715,E2 -6573.715} C_VEL
LIN {X 0,Y 488.008,Z 1083.101,A -85,B 0,C 180,E1 -6574.957,E2 -6574.957} C_VEL
LIN {X 0,Y 488.243,Z 1077.311,A -85,B 0,C 180,E1 -6576.198,E2 -6576.198} C_VEL
LIN {X 0,Y 488.339,Z 1071.17,A -85,B 0,C 180,E1 -6577.213,E2 -6577.213} C_VEL
LIN {X 0,Y 488.488,Z 1064.882,A -85,B 0,C 180,E1 -6578.064,E2 -6578.064} C_VEL
LIN {X 0,Y 488.767,Z 1057.407,A -85,B 0,C 180,E1 -6578.892,E2 -6578.892} C_VEL
LIN {X 0,Y 489.001,Z 1049.385,A -85,B 0,C 180,E1 -6579.618,E2 -6579.618} C_VEL
LIN {X 0,Y 489.33,Z 1039.352,A -85,B 0,C 180,E1 -6580.342,E2 -6580.342} C_VEL
LIN {X 0,Y 489.495,Z 1028.664,A -85,B 0,C 180,E1 -6580.914,E2 -6580.914} C_VEL
LIN {X 0,Y 489.705,Z 1018.588,A -85,B 0,C 180,E1 -6581.302,E2 -6581.302} C_VEL
LIN {X 0,Y 489.93,Z 1009.855,A -85,B 0,C 180,E1 -6581.533,E2 -6581.533} C_VEL
LIN {X 0,Y 490.145,Z 966.703,A -85,B 0,C 180,E1 -6582.206,E2 -6582.206} C_VEL
LIN {X 0,Y 490.062,Z 942.896,A -85,B 0,C 180,E1 -6582.556,E2 -6582.556} C_VEL
LIN {X 0,Y 488.654,Z 931.787,A -85,B 0,C 180,E1 -6582.786,E2 -6582.786} C_VEL
LIN {X 0,Y 489.06,Z 915.396,A -85,B 0,C 180,E1 -6585.845,E2 -6585.845} C_VEL
LIN {X 0,Y 489.567,Z 898.228,A -85,B 0,C 180,E1 -6589.087,E2 -6589.087} C_VEL
LIN {X 0,Y 490.057,Z 883.618,A -85,B 0,C 180,E1 -6591.893,E2 -6591.893} C_VEL
LIN {X 0,Y 489.53,Z 879.068,A -85,B 0,C 180,E1 -6592.807,E2 -6592.807} C_VEL
LIN {X 0,Y 488.727,Z 874.421,A -85,B 0,C 180,E1 -6593.8,E2 -6593.8} C_VEL
LIN {X 0,Y 488.672,Z 874.43,A -85,B 0,C 180,E1 -6597.401,E2 -6597.401} C_VEL
LIN {X 0,Y 488.649,Z 874.426,A -85,B 0,C 180,E1 -6600.351,E2 -6600.351} C_VEL
LIN {X 0,Y 488.706,Z 874.426,A -85,B 0,C 180,E1 -6603.479,E2 -6603.479} C_VEL
LIN {X 0,Y 488.64,Z 874.426,A -85,B 0,C 180,E1 -6606.348,E2 -6606.348} C_VEL
LIN {X 0,Y 488.663,Z 874.428,A -85,B 0,C 180,E1 -6609.258,E2 -6609.258} C_VEL
LIN {X 0,Y 488.645,Z 874.426,A -85,B 0,C 180,E1 -6612.531,E2 -6612.531} C_VEL
LIN {X 0,Y 488.693,Z 874.421,A -85,B 0,C 180,E1 -6615.197,E2 -6615.197} C_VEL
LIN {X 0,Y 488.64,Z 874.428,A -85,B 0,C 180,E1 -6618.578,E2 -6618.578} C_VEL
LIN {X 0,Y 488.641,Z 874.43,A -85,B 0,C 180,E1 -6621.797,E2 -6621.797} C_VEL
LIN {X 0,Y 488.71,Z 874.418,A -85,B 0,C 180,E1 -6625.055,E2 -6625.055} C_VEL
LIN {X 0,Y 488.683,Z 874.425,A -85,B 0,C 180,E1 -6628.05,E2 -6628.05} C_VEL
LIN {X 0,Y 488.658,Z 874.425,A -85,B 0,C 180,E1 -6631.32,E2 -6631.32} C_VEL
LIN {X 0,Y 488.665,Z 874.424,A -85,B 0,C 180,E1 -6633.523,E2 -6633.523} C_VEL
LIN {X 0,Y 488.652,Z 874.43,A -85,B 0,C 180,E1 -6636.253,E2 -6636.253} C_VEL
LIN {X 0,Y 488.712,Z 874.424,A -85,B 0,C 180,E1 -6639.187,E2 -6639.187} C_VEL
LIN {X 0,Y 488.766,Z 874.534,A -85,B 0,C 180,E1 -6641.753,E2 -6641.753} C_VEL
LIN {X 0,Y 489.013,Z 878.715,A -85,B 0,C 180,E1 -6642.865,E2 -6642.865} C_VEL
LIN {X 0,Y 488.686,Z 890.21,A -85,B 0,C 180,E1 -6645.849,E2 -6645.849} C_VEL
LIN {X 0,Y 488.553,Z 895.882,A -85,B 0,C 180,E1 -6647.301,E2 -6647.301} C_VEL
LIN {X 0,Y 490.3,Z 907.21,A -85,B 0,C 180,E1 -6647.526,E2 -6647.526} C_VEL
LIN {X 0,Y 489.876,Z 971.539,A -85,B 0,C 180,E1 -6648.519,E2 -6648.519} C_VEL
LIN {X 0,Y 489.713,Z 982.722,A -85,B 0,C 180,E1 -6648.829,E2 -6648.829} C_VEL
LIN {X 0,Y 489.457,Z 994.454,A -85,B 0,C 180,E1 -6649.347,E2 -6649.347} C_VEL
LIN {X 0,Y 489.256,Z 1003.186,A -85,B 0,C 180,E1 -6649.865,E2 -6649.865} C_VEL
LIN {X 0,Y 489.03,Z 1012.726,A -85,B 0,C 180,E1 -6650.592,E2 -6650.592} C_VEL
LIN {X 0,Y 488.695,Z 1022.318,A -85,B 0,C 180,E1 -6651.524,E2 -6651.524} C_VEL
LIN {X 0,Y 488.448,Z 1030.534,A -85,B 0,C 180,E1 -6652.56,E2 -6652.56} C_VEL
LIN {X 0,Y 488.3,Z 1036.697,A -85,B 0,C 180,E1 -6653.535,E2 -6653.535} C_VEL
LIN {X 0,Y 488.104,Z 1042.235,A -85,B 0,C 180,E1 -6654.63,E2 -6654.63} C_VEL
LIN {X 0,Y 488.067,Z 1046.983,A -85,B 0,C 180,E1 -6655.872,E2 -6655.872} C_VEL
LIN {X 0,Y 487.988,Z 1049.355,A -85,B 0,C 180,E1 -6656.698,E2 -6656.698} C_VEL
LIN {X 0,Y 487.924,Z 1051.162,A -85,B 0,C 180,E1 -6657.524,E2 -6657.524} C_VEL
LIN {X 0,Y 487.89,Z 1052.46,A -85,B 0,C 180,E1 -6658.349,E2 -6658.349} C_VEL
LIN {X 0,Y 487.831,Z 1053.258,A -85,B 0,C 180,E1 -6659.175,E2 -6659.175} C_VEL
LIN {X 0,Y 487.817,Z 1053.534,A -85,B 0,C 180,E1 -6660,E2 -6660} C_VEL
LIN {X 0,Y 487.832,Z 1053.288,A -85,B 0,C 180,E1 -6660.826,E2 -6660.826} C_VEL
LIN {X 0,Y 487.89,Z 1052.549,A -85,B 0,C 180,E1 -6661.651,E2 -6661.651} C_VEL
LIN {X 0,Y 487.912,Z 1051.318,A -85,B 0,C 180,E1 -6662.477,E2 -6662.477} C_VEL
LIN {X 0,Y 488.025,Z 1048.449,A -85,B 0,C 180,E1 -6663.716,E2 -6663.716} C_VEL
LIN {X 0,Y 488.003,Z 1044.301,A -85,B 0,C 180,E1 -6664.957,E2 -6664.957} C_VEL
LIN {X 0,Y 488.311,Z 1038.639,A -85,B 0,C 180,E1 -6666.197,E2 -6666.197} C_VEL
LIN {X 0,Y 488.359,Z 1032.664,A -85,B 0,C 180,E1 -6667.214,E2 -6667.214} C_VEL
LIN {X 0,Y 488.59,Z 1024.77,A -85,B 0,C 180,E1 -6668.271,E2 -6668.271} C_VEL
LIN {X 0,Y 488.921,Z 1016.03,A -85,B 0,C 180,E1 -6669.202,E2 -6669.202} C_VEL
LIN {X 0,Y 489.232,Z 1005.976,A -85,B 0,C 180,E1 -6670.031,E2 -6670.031} C_VEL
LIN {X 0,Y 489.439,Z 997.959,A -85,B 0,C 180,E1 -6670.55,E2 -6670.55} C_VEL
LIN {X 0,Y 489.596,Z 988.783,A -85,B 0,C 180,E1 -6671.017,E2 -6671.017} C_VEL
LIN {X 0,Y 489.779,Z 979.113,A -85,B 0,C 180,E1 -6671.38,E2 -6671.38} C_VEL
LIN {X 0,Y 489.954,Z 969.171,A -85,B 0,C 180,E1 -6671.626,E2 -6671.626} C_VEL
LIN {X 0,Y 490.137,Z 905.589,A -85,B 0,C 180,E1 -6672.595,E2 -6672.595} C_VEL
LIN {X 0,Y 488.483,Z 895.42,A -85,B 0,C 180,E1 -6672.812,E2 -6672.812} C_VEL
LIN {X 0,Y 488.788,Z 883.43,A -85,B 0,C 180,E1 -6675.855,E2 -6675.855} C_VEL
LIN {X 0,Y 488.916,Z 875.119,A -85,B 0,C 180,E1 -6677.987,E2 -6677.987} C_VEL
LIN {X 0,Y 488.778,Z 874.415,A -85,B 0,C 180,E1 -6678.194,E2 -6678.194} C_VEL
LIN {X 0,Y 488.7,Z 874.427,A -85,B 0,C 180,E1 -6681.072,E2 -6681.072} C_VEL
LIN {X 0,Y 488.66,Z 874.425,A -85,B 0,C 180,E1 -6683.748,E2 -6683.748} C_VEL
LIN {X 0,Y 488.669,Z 874.422,A -85,B 0,C 180,E1 -6686.478,E2 -6686.478} C_VEL
LIN {X 0,Y 488.661,Z 874.429,A -85,B 0,C 180,E1 -6689.275,E2 -6689.275} C_VEL
LIN {X 0,Y 488.686,Z 874.421,A -85,B 0,C 180,E1 -6692.149,E2 -6692.149} C_VEL
LIN {X 0,Y 488.707,Z 874.418,A -85,B 0,C 180,E1 -6695.117,E2 -6695.117} C_VEL
LIN {X 0,Y 488.651,Z 874.428,A -85,B 0,C 180,E1 -6698.203,E2 -6698.203} C_VEL
LIN {X 0,Y 488.645,Z 874.426,A -85,B 0,C 180,E1 -6701.423,E2 -6701.423} C_VEL
LIN {X 0,Y 488.698,Z 874.419,A -85,B 0,C 180,E1 -6704.804,E2 -6704.804} C_VEL
LIN {X 0,Y 488.65,Z 874.424,A -85,B 0,C 180,E1 -6707.47,E2 -6707.47} C_VEL
LIN {X 0,Y 488.669,Z 874.425,A -85,B 0,C 180,E1 -6710.743,E2 -6710.743} C_VEL
LIN {X 0,Y 488.647,Z 874.425,A -85,B 0,C 180,E1 -6713.712,E2 -6713.712} C_VEL
LIN {X 0,Y 487.987,Z 874.513,A -85,B 0,C 180,E1 -6714.4,E2 -6714.4} C_VEL
LIN {X 0,Y 485.167,Z 874.864,A -85,B 0,C 180,E1 -6715.518,E2 -6715.518} C_VEL
LIN {X 0,Y 482.776,Z 875.161,A -85,B 0,C 180,E1 -6716.419,E2 -6716.419} C_VEL
LIN {X 0,Y 481.738,Z 875.288,A -85,B 0,C 180,E1 -6717.115,E2 -6717.115} C_VEL
LIN {X 0,Y 481.647,Z 875.298,A -85,B 0,C 180,E1 -6717.35,E2 -6717.35} C_VEL
LIN {X 0,Y 481.603,Z 875.304,A -85,B 0,C 180,E1 -6720.254,E2 -6720.254} C_VEL
LIN {X 0,Y 481.651,Z 875.302,A -85,B 0,C 180,E1 -6723.106,E2 -6723.106} C_VEL
LIN {X 0,Y 481.645,Z 875.297,A -85,B 0,C 180,E1 -6725.885,E2 -6725.885} C_VEL
LIN {X 0,Y 481.686,Z 875.298,A -85,B 0,C 180,E1 -6729.035,E2 -6729.035} C_VEL
LIN {X 0,Y 481.667,Z 875.294,A -85,B 0,C 180,E1 -6732.157,E2 -6732.157} C_VEL
LIN {X 0,Y 481.742,Z 875.285,A -85,B 0,C 180,E1 -6734.776,E2 -6734.776} C_VEL
LIN {X 0,Y 481.718,Z 875.289,A -85,B 0,C 180,E1 -6738.214,E2 -6738.214} C_VEL
LIN {X 0,Y 481.716,Z 875.295,A -85,B 0,C 180,E1 -6741.611,E2 -6741.611} C_VEL
LIN {X 0,Y 481.775,Z 875.285,A -85,B 0,C 180,E1 -6744.139,E2 -6744.139} C_VEL
LIN {X 0,Y 481.901,Z 875.267,A -85,B 0,C 180,E1 -6747.493,E2 -6747.493} C_VEL
LIN {X 0,Y 481.913,Z 875.27,A -85,B 0,C 180,E1 -6750,E2 -6750} C_VEL
LIN {X 0,Y 481.9,Z 875.269,A -85,B 0,C 180,E1 -6752.508,E2 -6752.508} C_VEL
LIN {X 0,Y 481.775,Z 875.282,A -85,B 0,C 180,E1 -6755.861,E2 -6755.861} C_VEL
LIN {X 0,Y 481.716,Z 875.295,A -85,B 0,C 180,E1 -6758.389,E2 -6758.389} C_VEL
LIN {X 0,Y 481.719,Z 875.287,A -85,B 0,C 180,E1 -6761.786,E2 -6761.786} C_VEL
LIN {X 0,Y 481.695,Z 875.293,A -85,B 0,C 180,E1 -6765.226,E2 -6765.226} C_VEL
LIN {X 0,Y 481.676,Z 875.295,A -85,B 0,C 180,E1 -6768.485,E2 -6768.485} C_VEL
LIN {X 0,Y 481.64,Z 875.301,A -85,B 0,C 180,E1 -6771.395,E2 -6771.395} C_VEL
LIN {X 0,Y 481.62,Z 875.3,A -85,B 0,C 180,E1 -6774.116,E2 -6774.116} C_VEL
LIN {X 0,Y 481.646,Z 875.302,A -85,B 0,C 180,E1 -6777.114,E2 -6777.114} C_VEL
LIN {X 0,Y 481.604,Z 875.306,A -85,B 0,C 180,E1 -6779.746,E2 -6779.746} C_VEL
LIN {X 0,Y 481.635,Z 875.298,A -85,B 0,C 180,E1 -6782.677,E2 -6782.677} C_VEL
LIN {X 0,Y 481.643,Z 875.299,A -85,B 0,C 180,E1 -6785.2,E2 -6785.2} C_VEL
LIN {X 0,Y 481.623,Z 875.305,A -85,B 0,C 180,E1 -6788.001,E2 -6788.001} C_VEL
LIN {X 0,Y 481.607,Z 875.301,A -85,B 0,C 180,E1 -6791.047,E2 -6791.047} C_VEL
LIN {X 0,Y 481.654,Z 875.299,A -85,B 0,C 180,E1 -6794.458,E2 -6794.458} C_VEL
LIN {X 0,Y 481.615,Z 875.302,A -85,B 0,C 180,E1 -6796.856,E2 -6796.856} C_VEL
LIN {X 0,Y 481.631,Z 875.303,A -85,B 0,C 180,E1 -6800.054,E2 -6800.054} C_VEL
LIN {X 0,Y 481.604,Z 875.302,A -85,B 0,C 180,E1 -6803.25,E2 -6803.25} C_VEL
LIN {X 0,Y 481.675,Z 875.297,A -85,B 0,C 180,E1 -6806.327,E2 -6806.327} C_VEL
LIN {X 0,Y 481.614,Z 875.302,A -85,B 0,C 180,E1 -6809.426,E2 -6809.426} C_VEL
LIN {X 0,Y 481.645,Z 875.297,A -85,B 0,C 180,E1 -6812.164,E2 -6812.164} C_VEL
LIN {X 0,Y 481.669,Z 875.302,A -85,B 0,C 180,E1 -6814.967,E2 -6814.967} C_VEL
LIN {X 0,Y 481.64,Z 875.299,A -85,B 0,C 180,E1 -6817.704,E2 -6817.704} C_VEL
LIN {X 0,Y 481.66,Z 875.295,A -85,B 0,C 180,E1 -6820.391,E2 -6820.391} C_VEL
LIN {X 0,Y 481.658,Z 875.299,A -85,B 0,C 180,E1 -6823.032,E2 -6823.032} C_VEL
LIN {X 0,Y 481.661,Z 875.301,A -85,B 0,C 180,E1 -6825.637,E2 -6825.637} C_VEL
LIN {X 0,Y 481.717,Z 875.289,A -85,B 0,C 180,E1 -6828.214,E2 -6828.214} C_VEL
LIN {X 0,Y 481.714,Z 875.295,A -85,B 0,C 180,E1 -6831.61,E2 -6831.61} C_VEL
LIN {X 0,Y 481.773,Z 875.285,A -85,B 0,C 180,E1 -6834.139,E2 -6834.139} C_VEL
LIN {X 0,Y 481.899,Z 875.267,A -85,B 0,C 180,E1 -6837.492,E2 -6837.492} C_VEL
LIN {X 0,Y 481.911,Z 875.271,A -85,B 0,C 180,E1 -6840,E2 -6840} C_VEL
LIN {X 0,Y 481.898,Z 875.27,A -85,B 0,C 180,E1 -6842.507,E2 -6842.507} C_VEL
LIN {X 0,Y 481.772,Z 875.283,A -85,B 0,C 180,E1 -6845.861,E2 -6845.861} C_VEL
LIN {X 0,Y 481.713,Z 875.296,A -85,B 0,C 180,E1 -6848.389,E2 -6848.389} C_VEL
LIN {X 0,Y 481.716,Z 875.288,A -85,B 0,C 180,E1 -6851.785,E2 -6851.785} C_VEL
LIN {X 0,Y 481.698,Z 875.293,A -85,B 0,C 180,E1 -6855.225,E2 -6855.225} C_VEL
LIN {X 0,Y 481.672,Z 875.296,A -85,B 0,C 180,E1 -6858.484,E2 -6858.484} C_VEL
LIN {X 0,Y 481.637,Z 875.301,A -85,B 0,C 180,E1 -6861.395,E2 -6861.395} C_VEL
LIN {X 0,Y 481.616,Z 875.3,A -85,B 0,C 180,E1 -6864.116,E2 -6864.116} C_VEL
LIN {X 0,Y 481.642,Z 875.303,A -85,B 0,C 180,E1 -6867.114,E2 -6867.114} C_VEL
LIN {X 0,Y 481.6,Z 875.306,A -85,B 0,C 180,E1 -6869.746,E2 -6869.746} C_VEL
LIN {X 0,Y 481.63,Z 875.298,A -85,B 0,C 180,E1 -6872.677,E2 -6872.677} C_VEL
LIN {X 0,Y 481.639,Z 875.3,A -85,B 0,C 180,E1 -6875.2,E2 -6875.2} C_VEL
LIN {X 0,Y 481.619,Z 875.305,A -85,B 0,C 180,E1 -6878.001,E2 -6878.001} C_VEL
LIN {X 0,Y 481.603,Z 875.302,A -85,B 0,C 180,E1 -6881.047,E2 -6881.047} C_VEL
LIN {X 0,Y 481.649,Z 875.299,A -85,B 0,C 180,E1 -6884.458,E2 -6884.458} C_VEL
LIN {X 0,Y 481.611,Z 875.302,A -85,B 0,C 180,E1 -6886.855,E2 -6886.855} C_VEL
LIN {X 0,Y 481.626,Z 875.304,A -85,B 0,C 180,E1 -6890.054,E2 -6890.054} C_VEL
LIN {X 0,Y 481.599,Z 875.303,A -85,B 0,C 180,E1 -6893.25,E2 -6893.25} C_VEL
LIN {X 0,Y 481.67,Z 875.298,A -85,B 0,C 180,E1 -6896.327,E2 -6896.327} C_VEL
LIN {X 0,Y 481.609,Z 875.302,A -85,B 0,C 180,E1 -6899.426,E2 -6899.426} C_VEL
LIN {X 0,Y 481.64,Z 875.298,A -85,B 0,C 180,E1 -6902.164,E2 -6902.164} C_VEL
LIN {X 0,Y 481.664,Z 875.305,A -85,B 0,C 180,E1 -6904.967,E2 -6904.967} C_VEL
LIN {X 0,Y 481.704,Z 875.476,A -85,B 0,C 180,E1 -6905.945,E2 -6905.945} C_VEL
LIN {X 0,Y 483.164,Z 884.167,A -85,B 0,C 180,E1 -6907.778,E2 -6907.778} C_VEL
LIN {X 0,Y 482.705,Z 898.972,A -85,B 0,C 180,E1 -6910.678,E2 -6910.678} C_VEL
LIN {X 0,Y 482.131,Z 915.767,A -85,B 0,C 180,E1 -6913.921,E2 -6913.921} C_VEL
LIN {X 0,Y 481.652,Z 932.038,A -85,B 0,C 180,E1 -6917.047,E2 -6917.047} C_VEL
LIN {X 0,Y 483.262,Z 944.646,A -85,B 0,C 180,E1 -6917.291,E2 -6917.291} C_VEL
LIN {X 0,Y 483.049,Z 1005.977,A -85,B 0,C 180,E1 -6918.227,E2 -6918.227} C_VEL
LIN {X 0,Y 482.795,Z 1016.628,A -85,B 0,C 180,E1 -6918.48,E2 -6918.48} C_VEL
LIN {X 0,Y 482.622,Z 1025.942,A -85,B 0,C 180,E1 -6918.822,E2 -6918.822} C_VEL
LIN {X 0,Y 482.395,Z 1033.532,A -85,B 0,C 180,E1 -6919.188,E2 -6919.188} C_VEL
LIN {X 0,Y 482.191,Z 1042.096,A -85,B 0,C 180,E1 -6919.715,E2 -6919.715} C_VEL
LIN {X 0,Y 481.965,Z 1050.319,A -85,B 0,C 180,E1 -6920.346,E2 -6920.346} C_VEL
LIN {X 0,Y 481.692,Z 1058.125,A -85,B 0,C 180,E1 -6921.082,E2 -6921.082} C_VEL
LIN {X 0,Y 481.39,Z 1066.302,A -85,B 0,C 180,E1 -6922.028,E2 -6922.028} C_VEL
LIN {X 0,Y 481.216,Z 1073.472,A -85,B 0,C 180,E1 -6923.08,E2 -6923.08} C_VEL
LIN {X 0,Y 481.1,Z 1079.115,A -85,B 0,C 180,E1 -6924.131,E2 -6924.131} C_VEL
LIN {X 0,Y 480.9,Z 1084.352,A -85,B 0,C 180,E1 -6925.39,E2 -6925.39} C_VEL
LIN {X 0,Y 480.948,Z 1087.046,A -85,B 0,C 180,E1 -6926.229,E2 -6926.229} C_VEL
LIN {X 0,Y 480.827,Z 1089.982,A -85,B 0,C 180,E1 -6927.487,E2 -6927.487} C_VEL
LIN {X 0,Y 480.82,Z 1091.256,A -85,B 0,C 180,E1 -6928.325,E2 -6928.325} C_VEL
LIN {X 0,Y 480.756,Z 1092.044,A -85,B 0,C 180,E1 -6929.162,E2 -6929.162} C_VEL
LIN {X 0,Y 480.74,Z 1092.337,A -85,B 0,C 180,E1 -6930,E2 -6930} C_VEL
LIN {X 0,Y 480.756,Z 1092.036,A -85,B 0,C 180,E1 -6930.837,E2 -6930.837} C_VEL
LIN {X 0,Y 480.819,Z 1091.245,A -85,B 0,C 180,E1 -6931.675,E2 -6931.675} C_VEL
LIN {X 0,Y 480.826,Z 1089.962,A -85,B 0,C 180,E1 -6932.513,E2 -6932.513} C_VEL
LIN {X 0,Y 480.946,Z 1087.014,A -85,B 0,C 180,E1 -6933.77,E2 -6933.77} C_VEL
LIN {X 0,Y 480.942,Z 1082.757,A -85,B 0,C 180,E1 -6935.03,E2 -6935.03} C_VEL
LIN {X 0,Y 481.138,Z 1077.752,A -85,B 0,C 180,E1 -6936.138,E2 -6936.138} C_VEL
LIN {X 0,Y 481.291,Z 1070.615,A -85,B 0,C 180,E1 -6937.341,E2 -6937.341} C_VEL
LIN {X 0,Y 481.448,Z 1064.434,A -85,B 0,C 180,E1 -6938.182,E2 -6938.182} C_VEL
LIN {X 0,Y 481.733,Z 1056.917,A -85,B 0,C 180,E1 -6939.023,E2 -6939.023} C_VEL
LIN {X 0,Y 481.972,Z 1048.834,A -85,B 0,C 180,E1 -6939.759,E2 -6939.759} C_VEL
LIN {X 0,Y 482.314,Z 1038.723,A -85,B 0,C 180,E1 -6940.494,E2 -6940.494} C_VEL
LIN {X 0,Y 482.511,Z 1027.876,A -85,B 0,C 180,E1 -6941.074,E2 -6941.074} C_VEL
LIN {X 0,Y 482.73,Z 1018.465,A -85,B 0,C 180,E1 -6941.441,E2 -6941.441} C_VEL
LIN {X 0,Y 482.934,Z 1009.856,A -85,B 0,C 180,E1 -6941.676,E2 -6941.676} C_VEL
LIN {X 0,Y 483.149,Z 968.272,A -85,B 0,C 180,E1 -6942.346,E2 -6942.346} C_VEL
LIN {X 0,Y 483.095,Z 943.349,A -85,B 0,C 180,E1 -6942.721,E2 -6942.721} C_VEL
LIN {X 0,Y 481.648,Z 931.503,A -85,B 0,C 180,E1 -6942.964,E2 -6942.964} C_VEL
LIN {X 0,Y 482.045,Z 915.06,A -85,B 0,C 180,E1 -6946.082,E2 -6946.082} C_VEL
LIN {X 0,Y 482.577,Z 898.166,A -85,B 0,C 180,E1 -6949.327,E2 -6949.327} C_VEL
LIN {X 0,Y 483.084,Z 884.503,A -85,B 0,C 180,E1 -6952,E2 -6952} C_VEL
LIN {X 0,Y 482.3,Z 878.874,A -85,B 0,C 180,E1 -6953.169,E2 -6953.169} C_VEL
LIN {X 0,Y 481.671,Z 875.3,A -85,B 0,C 180,E1 -6953.948,E2 -6953.948} C_VEL
LIN {X 0,Y 481.639,Z 875.307,A -85,B 0,C 180,E1 -6957.114,E2 -6957.114} C_VEL
LIN {X 0,Y 481.597,Z 875.307,A -85,B 0,C 180,E1 -6959.747,E2 -6959.747} C_VEL
LIN {X 0,Y 481.643,Z 875.301,A -85,B 0,C 180,E1 -6962.676,E2 -6962.676} C_VEL
LIN {X 0,Y 481.646,Z 875.305,A -85,B 0,C 180,E1 -6965.202,E2 -6965.202} C_VEL
LIN {X 0,Y 481.616,Z 875.305,A -85,B 0,C 180,E1 -6968.002,E2 -6968.002} C_VEL
LIN {X 0,Y 481.601,Z 875.303,A -85,B 0,C 180,E1 -6971.047,E2 -6971.047} C_VEL
LIN {X 0,Y 481.647,Z 875.299,A -85,B 0,C 180,E1 -6974.459,E2 -6974.459} C_VEL
LIN {X 0,Y 481.609,Z 875.302,A -85,B 0,C 180,E1 -6976.856,E2 -6976.856} C_VEL
LIN {X 0,Y 481.625,Z 875.307,A -85,B 0,C 180,E1 -6980.055,E2 -6980.055} C_VEL
LIN {X 0,Y 481.598,Z 875.303,A -85,B 0,C 180,E1 -6983.251,E2 -6983.251} C_VEL
LIN {X 0,Y 481.669,Z 875.302,A -85,B 0,C 180,E1 -6986.327,E2 -6986.327} C_VEL
LIN {X 0,Y 481.608,Z 875.303,A -85,B 0,C 180,E1 -6989.426,E2 -6989.426} C_VEL
LIN {X 0,Y 481.639,Z 875.301,A -85,B 0,C 180,E1 -6992.165,E2 -6992.165} C_VEL
LIN {X 0,Y 481.662,Z 875.305,A -85,B 0,C 180,E1 -6994.967,E2 -6994.967} C_VEL
LIN {X 0,Y 481.633,Z 875.304,A -85,B 0,C 180,E1 -6997.704,E2 -6997.704} C_VEL
LIN {X 0,Y 481.654,Z 875.301,A -85,B 0,C 180,E1 -7000.391,E2 -7000.391} C_VEL
LIN {X 0,Y 481.713,Z 875.439,A -85,B 0,C 180,E1 -7001.628,E2 -7001.628} C_VEL
LIN {X 0,Y 481.981,Z 880.679,A -85,B 0,C 180,E1 -7003.045,E2 -7003.045} C_VEL
LIN {X 0,Y 481.673,Z 890.54,A -85,B 0,C 180,E1 -7005.639,E2 -7005.639} C_VEL
LIN {X 0,Y 481.54,Z 896.189,A -85,B 0,C 180,E1 -7007.108,E2 -7007.108} C_VEL
LIN {X 0,Y 483.384,Z 908.203,A -85,B 0,C 180,E1 -7007.36,E2 -7007.36} C_VEL
LIN {X 0,Y 482.903,Z 972.193,A -85,B 0,C 180,E1 -7008.377,E2 -7008.377} C_VEL
LIN {X 0,Y 482.741,Z 983.992,A -85,B 0,C 180,E1 -7008.719,E2 -7008.719} C_VEL
LIN {X 0,Y 482.483,Z 994.416,A -85,B 0,C 180,E1 -7009.191,E2 -7009.191} C_VEL
LIN {X 0,Y 482.272,Z 1003.19,A -85,B 0,C 180,E1 -7009.717,E2 -7009.717} C_VEL
LIN {X 0,Y 482.079,Z 1011.547,A -85,B 0,C 180,E1 -7010.349,E2 -7010.349} C_VEL
LIN {X 0,Y 481.789,Z 1019.435,A -85,B 0,C 180,E1 -7011.084,E2 -7011.084} C_VEL
LIN {X 0,Y 481.538,Z 1025.943,A -85,B 0,C 180,E1 -7011.819,E2 -7011.819} C_VEL
LIN {X 0,Y 481.37,Z 1032.269,A -85,B 0,C 180,E1 -7012.682,E2 -7012.682} C_VEL
LIN {X 0,Y 481.25,Z 1039.049,A -85,B 0,C 180,E1 -7013.829,E2 -7013.829} C_VEL
LIN {X 0,Y 480.943,Z 1044.249,A -85,B 0,C 180,E1 -7014.97,E2 -7014.97} C_VEL
LIN {X 0,Y 480.96,Z 1048.483,A -85,B 0,C 180,E1 -7016.23,E2 -7016.23} C_VEL
LIN {X 0,Y 480.838,Z 1051.429,A -85,B 0,C 180,E1 -7017.487,E2 -7017.487} C_VEL
LIN {X 0,Y 480.821,Z 1052.727,A -85,B 0,C 180,E1 -7018.325,E2 -7018.325} C_VEL
LIN {X 0,Y 480.757,Z 1053.536,A -85,B 0,C 180,E1 -7019.163,E2 -7019.163} C_VEL
LIN {X 0,Y 480.741,Z 1053.819,A -85,B 0,C 180,E1 -7020,E2 -7020} C_VEL
LIN {X 0,Y 480.758,Z 1053.557,A -85,B 0,C 180,E1 -7020.838,E2 -7020.838} C_VEL
LIN {X 0,Y 480.821,Z 1052.807,A -85,B 0,C 180,E1 -7021.676,E2 -7021.676} C_VEL
LIN {X 0,Y 480.827,Z 1051.571,A -85,B 0,C 180,E1 -7022.514,E2 -7022.514} C_VEL
LIN {X 0,Y 480.956,Z 1048.684,A -85,B 0,C 180,E1 -7023.771,E2 -7023.771} C_VEL
LIN {X 0,Y 480.938,Z 1044.531,A -85,B 0,C 180,E1 -7025.03,E2 -7025.03} C_VEL
LIN {X 0,Y 481.253,Z 1039.451,A -85,B 0,C 180,E1 -7026.171,E2 -7026.171} C_VEL
LIN {X 0,Y 481.32,Z 1032.815,A -85,B 0,C 180,E1 -7027.32,E2 -7027.32} C_VEL
LIN {X 0,Y 481.516,Z 1026.601,A -85,B 0,C 180,E1 -7028.182,E2 -7028.182} C_VEL
LIN {X 0,Y 481.82,Z 1018.193,A -85,B 0,C 180,E1 -7029.128,E2 -7029.128} C_VEL
LIN {X 0,Y 482.155,Z 1008.796,A -85,B 0,C 180,E1 -7029.968,E2 -7029.968} C_VEL
LIN {X 0,Y 482.398,Z 999.766,A -85,B 0,C 180,E1 -7030.599,E2 -7030.599} C_VEL
LIN {X 0,Y 482.604,Z 989.841,A -85,B 0,C 180,E1 -7031.126,E2 -7031.126} C_VEL
LIN {X 0,Y 482.756,Z 980.474,A -85,B 0,C 180,E1 -7031.494,E2 -7031.494} C_VEL
LIN {X 0,Y 482.976,Z 970.615,A -85,B 0,C 180,E1 -7031.755,E2 -7031.755} C_VEL
LIN {X 0,Y 483.162,Z 906.016,A -85,B 0,C 180,E1 -7032.773,E2 -7032.773} C_VEL
LIN {X 0,Y 481.451,Z 895.638,A -85,B 0,C 180,E1 -7033.003,E2 -7033.003} C_VEL
LIN {X 0,Y 481.784,Z 883.626,A -85,B 0,C 180,E1 -7036.091,E2 -7036.091} C_VEL
LIN {X 0,Y 481.789,Z 875.563,A -85,B 0,C 180,E1 -7038.187,E2 -7038.187} C_VEL
LIN {X 0,Y 481.734,Z 875.293,A -85,B 0,C 180,E1 -7038.388,E2 -7038.388} C_VEL
LIN {X 0,Y 481.637,Z 875.302,A -85,B 0,C 180,E1 -7041.396,E2 -7041.396} C_VEL
LIN {X 0,Y 481.621,Z 875.3,A -85,B 0,C 180,E1 -7044.117,E2 -7044.117} C_VEL
LIN {X 0,Y 481.643,Z 875.302,A -85,B 0,C 180,E1 -7047.115,E2 -7047.115} C_VEL
LIN {X 0,Y 481.601,Z 875.306,A -85,B 0,C 180,E1 -7049.747,E2 -7049.747} C_VEL
LIN {X 0,Y 481.647,Z 875.296,A -85,B 0,C 180,E1 -7052.677,E2 -7052.677} C_VEL
LIN {X 0,Y 481.651,Z 875.298,A -85,B 0,C 180,E1 -7055.202,E2 -7055.202} C_VEL
LIN {X 0,Y 481.627,Z 875.305,A -85,B 0,C 180,E1 -7058.003,E2 -7058.003} C_VEL
LIN {X 0,Y 481.606,Z 875.302,A -85,B 0,C 180,E1 -7061.048,E2 -7061.048} C_VEL
LIN {X 0,Y 481.652,Z 875.299,A -85,B 0,C 180,E1 -7064.459,E2 -7064.459} C_VEL
LIN {X 0,Y 481.614,Z 875.302,A -85,B 0,C 180,E1 -7066.856,E2 -7066.856} C_VEL
LIN {X 0,Y 481.63,Z 875.303,A -85,B 0,C 180,E1 -7070.055,E2 -7070.055} C_VEL
LIN {X 0,Y 481.606,Z 875.302,A -85,B 0,C 180,E1 -7073.251,E2 -7073.251} C_VEL
LIN {X 0,Y 481.674,Z 875.297,A -85,B 0,C 180,E1 -7076.327,E2 -7076.327} C_VEL
LIN {X 0,Y 481.647,Z 875.298,A -85,B 0,C 180,E1 -7077.35,E2 -7077.35} C_VEL
LIN {X 0,Y 480.964,Z 875.383,A -85,B 0,C 180,E1 -7078.048,E2 -7078.048} C_VEL
LIN {X 0,Y 478.105,Z 875.745,A -85,B 0,C 180,E1 -7079.182,E2 -7079.182} C_VEL
LIN {X 0,Y 475.695,Z 876.049,A -85,B 0,C 180,E1 -7080.096,E2 -7080.096} C_VEL
LIN {X 0,Y 474.659,Z 876.176,A -85,B 0,C 180,E1 -7080.801,E2 -7080.801} C_VEL
LIN {X 0,Y 474.574,Z 876.183,A -85,B 0,C 180,E1 -7081.04,E2 -7081.04} C_VEL
LIN {X 0,Y 474.574,Z 876.179,A -85,B 0,C 180,E1 -7083.623,E2 -7083.623} C_VEL
LIN {X 0,Y 474.601,Z 876.177,A -85,B 0,C 180,E1 -7086.653,E2 -7086.653} C_VEL
LIN {X 0,Y 474.653,Z 876.176,A -85,B 0,C 180,E1 -7089.185,E2 -7089.185} C_VEL
LIN {X 0,Y 474.623,Z 876.173,A -85,B 0,C 180,E1 -7091.883,E2 -7091.883} C_VEL
LIN {X 0,Y 474.701,Z 876.162,A -85,B 0,C 180,E1 -7094.545,E2 -7094.545} C_VEL
LIN {X 0,Y 474.681,Z 876.167,A -85,B 0,C 180,E1 -7098.037,E2 -7098.037} C_VEL
LIN {X 0,Y 474.664,Z 876.171,A -85,B 0,C 180,E1 -7101.485,E2 -7101.485} C_VEL
LIN {X 0,Y 474.739,Z 876.162,A -85,B 0,C 180,E1 -7104.052,E2 -7104.052} C_VEL
LIN {X 0,Y 474.842,Z 876.146,A -85,B 0,C 180,E1 -7107.455,E2 -7107.455} C_VEL
LIN {X 0,Y 474.883,Z 876.146,A -85,B 0,C 180,E1 -7110,E2 -7110} C_VEL
LIN {X 0,Y 474.84,Z 876.148,A -85,B 0,C 180,E1 -7112.545,E2 -7112.545} C_VEL
LIN {X 0,Y 474.739,Z 876.16,A -85,B 0,C 180,E1 -7115.948,E2 -7115.948} C_VEL
LIN {X 0,Y 474.665,Z 876.174,A -85,B 0,C 180,E1 -7118.515,E2 -7118.515} C_VEL
LIN {X 0,Y 474.681,Z 876.165,A -85,B 0,C 180,E1 -7121.963,E2 -7121.963} C_VEL
LIN {X 0,Y 474.655,Z 876.169,A -85,B 0,C 180,E1 -7125.457,E2 -7125.457} C_VEL
LIN {X 0,Y 474.633,Z 876.174,A -85,B 0,C 180,E1 -7128.617,E2 -7128.617} C_VEL
LIN {X 0,Y 474.623,Z 876.179,A -85,B 0,C 180,E1 -7131.111,E2 -7131.111} C_VEL
LIN {X 0,Y 474.586,Z 876.177,A -85,B 0,C 180,E1 -7134.497,E2 -7134.497} C_VEL
LIN {X 0,Y 474.597,Z 876.183,A -85,B 0,C 180,E1 -7137.327,E2 -7137.327} C_VEL
LIN {X 0,Y 474.553,Z 876.181,A -85,B 0,C 180,E1 -7140.234,E2 -7140.234} C_VEL
LIN {X 0,Y 474.602,Z 876.178,A -85,B 0,C 180,E1 -7143.224,E2 -7143.224} C_VEL
LIN {X 0,Y 474.568,Z 876.18,A -85,B 0,C 180,E1 -7146.326,E2 -7146.326} C_VEL
LIN {X 0,Y 474.6,Z 876.178,A -85,B 0,C 180,E1 -7149.551,E2 -7149.551} C_VEL
LIN {X 0,Y 474.569,Z 876.178,A -85,B 0,C 180,E1 -7152.94,E2 -7152.94} C_VEL
LIN {X 0,Y 474.602,Z 876.179,A -85,B 0,C 180,E1 -7155.893,E2 -7155.893} C_VEL
LIN {X 0,Y 474.584,Z 876.177,A -85,B 0,C 180,E1 -7159.047,E2 -7159.047} C_VEL
LIN {X 0,Y 474.585,Z 876.177,A -85,B 0,C 180,E1 -7161.708,E2 -7161.708} C_VEL
LIN {X 0,Y 474.613,Z 876.178,A -85,B 0,C 180,E1 -7164.724,E2 -7164.724} C_VEL
LIN {X 0,Y 474.62,Z 876.172,A -85,B 0,C 180,E1 -7167.786,E2 -7167.786} C_VEL
LIN {X 0,Y 474.579,Z 876.184,A -85,B 0,C 180,E1 -7170.895,E2 -7170.895} C_VEL
LIN {X 0,Y 474.574,Z 876.178,A -85,B 0,C 180,E1 -7173.623,E2 -7173.623} C_VEL
LIN {X 0,Y 474.601,Z 876.177,A -85,B 0,C 180,E1 -7176.652,E2 -7176.652} C_VEL
LIN {X 0,Y 474.653,Z 876.176,A -85,B 0,C 180,E1 -7179.184,E2 -7179.184} C_VEL
LIN {X 0,Y 474.622,Z 876.173,A -85,B 0,C 180,E1 -7181.882,E2 -7181.882} C_VEL
LIN {X 0,Y 474.656,Z 876.167,A -85,B 0,C 180,E1 -7184.542,E2 -7184.542} C_VEL
LIN {X 0,Y 474.679,Z 876.167,A -85,B 0,C 180,E1 -7188.036,E2 -7188.036} C_VEL
LIN {X 0,Y 474.663,Z 876.172,A -85,B 0,C 180,E1 -7191.485,E2 -7191.485} C_VEL
LIN {X 0,Y 474.737,Z 876.162,A -85,B 0,C 180,E1 -7194.051,E2 -7194.051} C_VEL
LIN {X 0,Y 474.839,Z 876.146,A -85,B 0,C 180,E1 -7197.455,E2 -7197.455} C_VEL
LIN {X 0,Y 474.881,Z 876.147,A -85,B 0,C 180,E1 -7200,E2 -7200} C_VEL
LIN {X 0,Y 474.838,Z 876.148,A -85,B 0,C 180,E1 -7202.545,E2 -7202.545} C_VEL
LIN {X 0,Y 474.736,Z 876.16,A -85,B 0,C 180,E1 -7205.948,E2 -7205.948} C_VEL
LIN {X 0,Y 474.662,Z 876.175,A -85,B 0,C 180,E1 -7208.514,E2 -7208.514} C_VEL
LIN {X 0,Y 474.678,Z 876.165,A -85,B 0,C 180,E1 -7211.963,E2 -7211.963} C_VEL
LIN {X 0,Y 474.654,Z 876.169,A -85,B 0,C 180,E1 -7215.457,E2 -7215.457} C_VEL
LIN {X 0,Y 474.629,Z 876.175,A -85,B 0,C 180,E1 -7218.617,E2 -7218.617} C_VEL
LIN {X 0,Y 474.619,Z 876.179,A -85,B 0,C 180,E1 -7221.11,E2 -7221.11} C_VEL
LIN {X 0,Y 474.582,Z 876.177,A -85,B 0,C 180,E1 -7224.497,E2 -7224.497} C_VEL
LIN {X 0,Y 474.593,Z 876.183,A -85,B 0,C 180,E1 -7227.326,E2 -7227.326} C_VEL
LIN {X 0,Y 474.549,Z 876.181,A -85,B 0,C 180,E1 -7230.234,E2 -7230.234} C_VEL
LIN {X 0,Y 474.598,Z 876.178,A -85,B 0,C 180,E1 -7233.223,E2 -7233.223} C_VEL
LIN {X 0,Y 474.564,Z 876.18,A -85,B 0,C 180,E1 -7236.325,E2 -7236.325} C_VEL
LIN {X 0,Y 474.596,Z 876.179,A -85,B 0,C 180,E1 -7239.55,E2 -7239.55} C_VEL
LIN {X 0,Y 474.565,Z 876.179,A -85,B 0,C 180,E1 -7242.94,E2 -7242.94} C_VEL
LIN {X 0,Y 474.597,Z 876.18,A -85,B 0,C 180,E1 -7245.893,E2 -7245.893} C_VEL
LIN {X 0,Y 474.579,Z 876.177,A -85,B 0,C 180,E1 -7249.047,E2 -7249.047} C_VEL
LIN {X 0,Y 474.581,Z 876.177,A -85,B 0,C 180,E1 -7251.708,E2 -7251.708} C_VEL
